bInterruptStarted S= bInterrupt AND astMotionStage[1].bBusy AND astMotionStage[2].bBusy AND astMotionStage[3].bBusy;
fbMove(
    astMotionStage:=astMotionStage,
    astPositionState:=astGoalPositions,
    nActiveMotorCount:=3,
    bExecute:=NOT bInterruptStarted,
);
IF fbMove.bDone OR tonTimer.Q OR (bInterruptStarted AND NOT fbMove.bBusy) THEN
    IF bInterrupt THEN
        AssertFalse(
            fbMove.bAtState,
            Message:='Should have been interrupted, but made it to the goal',
        );
    ELSE
        AssertTrue(
            fbMove.bAtState,
            Message:='Did not end at the state',
        );
        FOR nIter := 1 TO 3 DO
            AssertEquals_LREAL(
                Expected:=astGoalPositions[nIter].fPosition,
                Actual:=astMotionStage[nIter].stAxisStatus.fActPosition,
                Delta:=0.01,
                Message:='Did not reach the goal state',
            );
        END_FOR

    END_IF
    AssertFalse(
        fbMove.bBusy,
        Message:='Was busy while done',
    );
    AssertFalse(
        fbMove.bError,
        Message:='Should not end in error',
    );

    bOneTestDone := TRUE;
    TEST_FINISHED();
END_IF
END_METHOD

END_FUNCTION_BLOCK

// Tests/FB_PositionStateND_Test
FUNCTION_BLOCK FB_PositionStateND_Test EXTENDS FB_MotorTestSuite
(*
    Sanity checks for the following:
    - FB_PositionState1D
    - FB_PositionState2D
    - FB_PositionState3D
    The internals have already been tested, but we need to make sure that
    they've been put together at least somewhat sensibly.
    This FB will simply use each FB to move and check the results.

    Additional tests:
    - Regression test for issue #197 (input deadlock)
*)
VAR
    stMotionStage1: ST_MotionStage;
    stMotionStage2: ST_MotionStage;
    stMotionStage3: ST_MotionStage;
    astPositionState1: ARRAY[1..GeneralConstants.MAX_STATES] OF ST_PositionState;
    astPositionState2: ARRAY[1..GeneralConstants.MAX_STATES] OF ST_PositionState;
    astPositionState3: ARRAY[1..GeneralConstants.MAX_STATES] OF ST_PositionState;
    afbInternal: ARRAY[1..3] OF ARRAY[1..3] OF FB_PositionStateInternal;
    afbMotionStage: ARRAY[1..3] OF FB_MotionStage;

    fb_Move1D: FB_PositionState1D;
    fb_Move2D: FB_PositionState2D;
    fb_Move3D: FB_PositionState3D;

    nTestCounter: UINT;
    bOneTestDone: BOOL;
    fTestStartPos: LREAL;
    tonTimer: TON;
    nIter: DINT;
    bStatesReady: BOOL;

    eSetPos: E_TestStates;
    eGetPos: E_TestStates;
END_VAR


bStatesReady := TRUE;
FOR nIter := 1 TO 3 DO;
    astPositionState1[nIter].fPosition := nIter;
    astPositionState1[nIter].fDelta := 1;
    astPositionState1[nIter].fVelocity := 100;
    astPositionState2[nIter].fPosition := 10 + nIter;
    astPositionState2[nIter].fDelta := 1;
    astPositionState2[nIter].fVelocity := 100;
    astPositionState3[nIter].fPosition := 20 + nIter;
    astPositionState3[nIter].fDelta := 1;
    astPositionState3[nIter].fVelocity := 100;
    afbInternal[nIter][1](
        stMotionStage:=stMotionStage1,
        stPositionState:=astPositionState1[nIter],
    );
    afbInternal[nIter][2](
        stMotionStage:=stMotionStage2,
        stPositionState:=astPositionState2[nIter],
    );
    afbInternal[nIter][3](
        stMotionStage:=stMotionStage3,
        stPositionState:=astPositionState3[nIter],
    );
    SetGoodState(astPositionState1[nIter]);
    SetGoodState(astPositionState2[nIter]);
    SetGoodState(astPositionState3[nIter]);
    bStatesReady := bStatesReady AND astPositionState1[nIter].bUpdated;
    bStatesReady := bStatesReady AND astPositionState2[nIter].bUpdated;
    bStatesReady := bStatesReady AND astPositionState3[nIter].bUpdated;
END_FOR
SetEnables(stMotionStage1);
SetEnables(stMotionStage2);
SetEnables(stMotionStage3);
afbMotionStage[1](stMotionStage:=stMotionStage1);
afbMotionStage[2](stMotionStage:=stMotionStage2);
afbMotionStage[3](stMotionStage:=stMotionStage3);

IF bStatesReady AND nTestCounter = 0 THEN
    // Don't run any tests until the states are ready
    nTestCounter := 1;
    // Run all the motion FBs for one cycle to warm them up
    fb_Move1D(
        stMotionStage:=stMotionStage1,
        astPositionState:=astPositionState1,
        eEnumSet:=eSetPos,
        eEnumGet:=eGetPos,
        bEnable:=TRUE,
    );
    fb_Move2D(
        stMotionStage1:=stMotionStage1,
        stMotionStage2:=stMotionStage2,
        astPositionState1:=astPositionState1,
        astPositionState2:=astPositionState2,
        eEnumSet:=eSetPos,
        eEnumGet:=eGetPos,
        bEnable:=TRUE,
    );
    fb_Move3D(
        stMotionStage1:=stMotionStage1,
        stMotionStage2:=stMotionStage2,
        stMotionStage3:=stMotionStage3,
        astPositionState1:=astPositionState1,
        astPositionState2:=astPositionState2,
        astPositionState3:=astPositionState3,
        eEnumSet:=eSetPos,
        eEnumGet:=eGetPos,
        bEnable:=TRUE,
    );
END_IF

Test1D(1, E_TestStates.OUT);
Test1D(2, E_TestStates.TARGET1);
Test1D(3, E_TestStates.TARGET2);
Test2D(4, E_TestStates.OUT);
Test2D(5, E_TestStates.TARGET1);
Test2D(6, E_TestStates.TARGET2);
Test3D(7, E_TestStates.OUT);
Test3D(8, E_TestStates.TARGET1);
Test3D(9, E_TestStates.TARGET2);
TestInputDeadlock(10);

IF bOneTestDone THEN
    bOneTestDone := FALSE;
    nTestCounter := nTestCounter + 1;
    tonTimer(IN:=FALSE);
END_IF
// Use this timer to time out any tests that stall
tonTimer(
    IN:=bStatesReady,
    PT:=T#5s,
);

METHOD Test1D
VAR_INPUT
    nTestID: UINT;
    nState: E_TestStates;
END_VAR
VAR_INST
    nLocalInit: BOOL;
END_VAR

TEST(CONCAT('Test1D_state', DINT_TO_STRING(nState)));
IF nTestCounter <> nTestID THEN
    RETURN;
END_IF

IF NOT nLocalInit THEN
    eSetPos := nState;
    nLocalInit := TRUE;
END_IF

fb_Move1D(
    stMotionStage:=stMotionStage1,
    astPositionState:=astPositionState1,
    eEnumSet:=eSetPos,
    eEnumGet:=eGetPos,
    bEnable:=TRUE,
);
IF tonTimer.Q OR fb_Move1D.stPlcToEpics.bDone THEN
    AssertTrue(
        Condition:=fb_Move1D.stPlcToEpics.bDone,
        Message:='Done should be True after move',
    );
    AssertFalse(
        Condition:=fb_Move1D.stPlcToEpics.bBusy,
        Message:='Busy should be False after move',
    );
    AssertFalse(
        Condition:=fb_Move1D.stPlcToEpics.bError,
        Message:='Error should be False after move',
    );
    AssertEquals_DINT(
        Expected:=nState,
        Actual:=eGetPos,
        Message:='Did not get to the input state',
    );
    AssertEquals_LREAL(
        Expected:=astPositionState1[nState].fPosition,
        Actual:=stMotionStage1.stAxisStatus.fActPosition,
        Delta:=0.1,
        Message:='Did not get to the input state position',
    );
    fb_Move1D.stEpicsToPlc.bReset := TRUE;
    fb_Move1D(
        stMotionStage:=stMotionStage1,
        astPositionState:=astPositionState1,
        eEnumSet:=eSetPos,
        eEnumGet:=eGetPos,
        bEnable:=TRUE,
    );
    bOneTestDone := TRUE;
    nLocalInit := FALSE;
    TEST_FINISHED();
END_IF
END_METHOD

METHOD Test2D
VAR_INPUT
    nTestID: UINT;
    nState: E_TestStates;
END_VAR
VAR_INST
    nLocalInit: BOOL;
END_VAR

TEST(CONCAT('Test2D_state', DINT_TO_STRING(nState)));
IF nTestCounter <> nTestID THEN
    RETURN;
END_IF

IF NOT nLocalInit THEN
    eSetPos := nState;
    nLocalInit := TRUE;
END_IF

fb_Move2D(
    stMotionStage1:=stMotionStage1,
    stMotionStage2:=stMotionStage2,
    astPositionState1:=astPositionState1,
    astPositionState2:=astPositionState2,
    eEnumSet:=eSetPos,
    eEnumGet:=eGetPos,
    bEnable:=TRUE,
);
IF tonTimer.Q OR fb_Move2D.stPlcToEpics.bDone THEN
    AssertTrue(
        Condition:=fb_Move2D.stPlcToEpics.bDone,
        Message:='Done should be True after move',
    );
    AssertFalse(
        Condition:=fb_Move2D.stPlcToEpics.bBusy,
        Message:='Busy should be False after move',
    );
    AssertFalse(
        Condition:=fb_Move2D.stPlcToEpics.bError,
        Message:='Error should be False after move',
    );
    AssertEquals_DINT(
        Expected:=nState,
        Actual:=eGetPos,
        Message:='Did not get to the input state',
    );
    AssertEquals_LREAL(
        Expected:=astPositionState1[nState].fPosition,
        Actual:=stMotionStage1.stAxisStatus.fActPosition,
        Delta:=0.1,
        Message:='Did not get to the input state position for stage 1',
    );
    AssertEquals_LREAL(
        Expected:=astPositionState2[nState].fPosition,
        Actual:=stMotionStage2.stAxisStatus.fActPosition,
        Delta:=0.1,
        Message:='Did not get to the input state position for stage 2',
    );
    fb_Move2D.stEpicsToPlc.bReset := TRUE;
    fb_Move2D(
        stMotionStage1:=stMotionStage1,
        stMotionStage2:=stMotionStage2,
        astPositionState1:=astPositionState1,
        astPositionState2:=astPositionState2,
        eEnumSet:=eSetPos,
        eEnumGet:=eGetPos,
        bEnable:=TRUE,
    );
    bOneTestDone := TRUE;
    nLocalInit := FALSE;
    TEST_FINISHED();
END_IF
END_METHOD

METHOD Test3D
VAR_INPUT
    nTestID: UINT;
    nState: E_TestStates;
END_VAR
VAR_INST
    nLocalInit: BOOL;
END_VAR

TEST(CONCAT('Test3D_state', DINT_TO_STRING(nState)));
IF nTestCounter <> nTestID THEN
    RETURN;
END_IF

IF NOT nLocalInit THEN
    eSetPos := nState;
    nLocalInit := TRUE;
END_IF

fb_Move3D(
    stMotionStage1:=stMotionStage1,
    stMotionStage2:=stMotionStage2,
    stMotionStage3:=stMotionStage3,
    astPositionState1:=astPositionState1,
    astPositionState2:=astPositionState2,
    astPositionState3:=astPositionState3,
    eEnumSet:=eSetPos,
    eEnumGet:=eGetPos,
    bEnable:=TRUE,
);
IF tonTimer.Q OR fb_Move3D.stPlcToEpics.bDone THEN
    AssertTrue(
        Condition:=fb_Move3D.stPlcToEpics.bDone,
        Message:='Done should be True after move',
    );
    AssertFalse(
        Condition:=fb_Move3D.stPlcToEpics.bBusy,
        Message:='Busy should be False after move',
    );
    AssertFalse(
        Condition:=fb_Move3D.stPlcToEpics.bError,
        Message:='Error should be False after move',
    );
    AssertEquals_DINT(
        Expected:=nState,
        Actual:=eGetPos,
        Message:='Did not get to the input state',
    );
    AssertEquals_LREAL(
        Expected:=astPositionState1[nState].fPosition,
        Actual:=stMotionStage1.stAxisStatus.fActPosition,
        Delta:=0.1,
        Message:='Did not get to the input state position for stage 1',
    );
    AssertEquals_LREAL(
        Expected:=astPositionState2[nState].fPosition,
        Actual:=stMotionStage2.stAxisStatus.fActPosition,
        Delta:=0.1,
        Message:='Did not get to the input state position for stage 2',
    );
    AssertEquals_LREAL(
        Expected:=astPositionState3[nState].fPosition,
        Actual:=stMotionStage3.stAxisStatus.fActPosition,
        Delta:=0.1,
        Message:='Did not get to the input state position for stage 3',
    );
    fb_Move3D.stEpicsToPlc.bReset := TRUE;
    fb_Move3D(
        stMotionStage1:=stMotionStage1,
        stMotionStage2:=stMotionStage2,
        stMotionStage3:=stMotionStage3,
        astPositionState1:=astPositionState1,
        astPositionState2:=astPositionState2,
        astPositionState3:=astPositionState3,
        eEnumSet:=eSetPos,
        eEnumGet:=eGetPos,
        bEnable:=TRUE,
    );
    bOneTestDone := TRUE;
    nLocalInit := FALSE;
    TEST_FINISHED();
END_IF
END_METHOD

METHOD TestInputDeadlock
(*
    Regression test for issue #197

    How to reproduce the issue:
    1. Get the function block into any motion error
    2. Ask for a move while in the error state

    Then, the state mover never moves again.

    To test we will follow steps 1 and 2, then reset the error, then move.

    With our fix, our second attempt at the move (after an error reset) will succeed.
    Our first attempt will fail regardless, since you cannot move a motor that is in an error state.

    Without our fix, the motor could never be moved ever again and this move will time out.
*)
VAR_INPUT
    nTestID: UINT;
END_VAR
VAR_INST
    nTestStep: UINT := 1;
    eNewGoal: E_TestStates;
END_VAR

TEST('TestInputDeadlock');
IF nTestCounter <> nTestID THEN
    RETURN;
END_IF

CASE nTestStep OF
    // Step 1: Normal move
    1:
        // Normal move: pick any other state
        IF eGetPos = E_TestStates.OUT THEN
            eNewGoal := E_TestStates.TARGET1;
        ELSE
            eNewGoal := E_TestStates.OUT;
        END_IF
        eSetPos := eNewGoal;
        nTestStep := 2;
    // Step 2: Cause a motion error. Easiest is to just set bError to TRUE during a move.
    2:
        // Cause the error if it's time
        IF stMotionStage1.bBusy THEN
            stMotionStage1.bError := TRUE;
            stMotionStage1.nErrorId := 16#4FFF;
        ELSIF stMotionStage1.bError THEN
            nTestStep := 3;
        END_IF
     // Step 3: another normal move. This should get us into the potential bugged state.
     3:
        eSetPos := eNewGoal;
        nTestStep := 4;
    // Step 4: reset the error, which will allow fixed versions of the code to resume normal operations.
    4:
        fb_Move1D.stEpicsToPlc.bReset := TRUE;
        IF NOT stMotionStage1.bError THEN
            nTestStep := 5;
        END_IF
    // Step 5: last normal move, which will succeed if we fixed the bug.
    5:
        eSetPos := eNewGoal;
        IF eGetPos = E_TestStates.Unknown THEN
            nTestStep := 6;
        END_IF
    // Step 6: wait for the move to finish
    6:
        IF eGetPos = eNewGoal THEN
            nTestStep := 7;
        END_IF
END_CASE

fb_Move1D(
    stMotionStage:=stMotionStage1,
    astPositionState:=astPositionState1,
    eEnumSet:=eSetPos,
    eEnumGet:=eGetPos,
    bEnable:=TRUE,
);

// Timeout and checks
IF tonTimer.Q OR nTestStep = 7 THEN
    AssertFalse(
        tonTimer.Q,
        'Timeout in deadlock test',
    );
    AssertEquals_UINT(
        Expected:=eNewGoal,
        Actual:=eGetPos,
        'Did not reach a goal state in deadlock test',
    );
    fb_Move1D.stEpicsToPlc.bReset := TRUE;
    fb_Move1D(
        stMotionStage:=stMotionStage1,
        astPositionState:=astPositionState1,
        eEnumSet:=eSetPos,
        eEnumGet:=eGetPos,
        bEnable:=TRUE,
    );
    bOneTestDone := TRUE;
    TEST_FINISHED();
END_IF
END_METHOD

END_FUNCTION_BLOCK

// Tests/FB_PositionStatePMPSND_Test
FUNCTION_BLOCK FB_PositionStatePMPSND_Test EXTENDS FB_MotorTestSuite
(*
    Sanity checks for the following:
    - FB_PositionStatePMPS1D
    - FB_PositionStatePMPS2D
    - FB_PositionStatePMPS3D
    The internals have already been tested, but we need to make sure that
    they've been put together at least somewhat sensibly.
    This FB will simply use each FB to move and check the results.
    In addition to reaching the goals, we need to check the beam assertions
    and the pmps limit enables.
*)
VAR
    stMotionStage1: ST_MotionStage;
    stMotionStage2: ST_MotionStage;
    stMotionStage3: ST_MotionStage;
    astPositionState1: ARRAY[1..GeneralConstants.MAX_STATES] OF ST_PositionState;
    astPositionState2: ARRAY[1..GeneralConstants.MAX_STATES] OF ST_PositionState;
    astPositionState3: ARRAY[1..GeneralConstants.MAX_STATES] OF ST_PositionState;
    afbInternal: ARRAY[1..3] OF ARRAY[1..3] OF FB_PositionStateInternal;
    afbMotionStage: ARRAY[1..3] OF FB_MotionStage;

    astBeam: ARRAY[0..3] OF ST_DbStateParams;

    fb_Move1D: FB_PositionStatePMPS1D;
    fb_Move2D: FB_PositionStatePMPS2D;
    fb_Move3D: FB_PositionStatePMPS3D;

    nTestCounter: UINT;
    bOneTestDone: BOOL;
    fTestStartPos: LREAL;
    tonTimer: TON;
    nIter: DINT;
    bStatesReady: BOOL;

    eSetPos: E_TestStates;
    eGetPos: E_TestStates;

    fbArbiter1D: FB_Arbiter(1);
    fbArbiter2D: FB_Arbiter(2);
    fbArbiter3D: FB_Arbiter(3);

    fbSubSysIO1D: FB_DummyArbIO;
    fbSubSysIO2D: FB_DummyArbIO;
    fbSubSysIO3D: FB_DummyArbIO;

    jsonHelper: FB_PMPSJsonTestHelper;
END_VAR


bStatesReady := TRUE;
FOR nIter := 1 TO 3 DO;
    astPositionState1[nIter].fPosition := nIter;
    astPositionState1[nIter].fDelta := 0.5;
    astPositionState1[nIter].fVelocity := 100;
    SetGoodState(astPositionState1[nIter]);
    astPositionState2[nIter].fPosition := 10 + nIter;
    astPositionState2[nIter].fDelta := 0.5;
    astPositionState2[nIter].fVelocity := 100;
    SetGoodState(astPositionState2[nIter]);
    astPositionState3[nIter].fPosition := 20 + nIter;
    astPositionState3[nIter].fDelta := 0.5;
    astPositionState3[nIter].fVelocity := 100;
    SetGoodState(astPositionState3[nIter]);
    afbInternal[nIter][1](
        stMotionStage:=stMotionStage1,
        stPositionState:=astPositionState1[nIter],
    );
    afbInternal[nIter][2](
        stMotionStage:=stMotionStage2,
        stPositionState:=astPositionState2[nIter],
    );
    afbInternal[nIter][3](
        stMotionStage:=stMotionStage3,
        stPositionState:=astPositionState3[nIter],
    );
    bStatesReady := bStatesReady AND astPositionState1[nIter].bUpdated;
    bStatesReady := bStatesReady AND astPositionState2[nIter].bUpdated;
    bStatesReady := bStatesReady AND astPositionState3[nIter].bUpdated;
END_FOR
SetEnablesPMPS(stMotionStage1);
SetEnablesPMPS(stMotionStage2);
SetEnablesPMPS(stMotionStage3);
IF nTestCounter <= 3 THEN
    // Startup tests, make sure the motor is enabled so we can inspect MC_Power's output
    // Otherwise we can't snoop on the PlcToNc control DWORD since this is all 0's if disabled
    // When enabled, some of the other bits go to 1 to represent directional enables
    stMotionStage1.nEnableMode := E_StageEnableMode.ALWAYS;
    stMotionStage2.nEnableMode := E_StageEnableMode.ALWAYS;
    stMotionStage3.nEnableMode := E_StageEnableMode.ALWAYS;
ELSE
    // Otherwise, make sure the most complicated mode (and the default) works
    stMotionStage1.nEnableMode := E_StageEnableMode.DURING_MOTION;
    stMotionStage2.nEnableMode := E_StageEnableMode.DURING_MOTION;
    stMotionStage3.nEnableMode := E_StageEnableMode.DURING_MOTION;
END_IF
afbMotionStage[1](stMotionStage:=stMotionStage1);
afbMotionStage[2](stMotionStage:=stMotionStage2);
afbMotionStage[3](stMotionStage:=stMotionStage3);

astBeam[E_TestStates.Unknown].stBeamParams := PMPS_GVL.cst0RateBeam;
astBeam[E_TestStates.Unknown].nRequestAssertionID := 1;
astBeam[E_TestStates.Unknown].sPmpsState := 'trans';
astBeam[E_TestStates.OUT].stBeamParams := PMPS_GVL.cstFullBeam;
astBeam[E_TestStates.OUT].nRequestAssertionID := 2;
astBeam[E_TestStates.OUT].sPmpsState := 'out';
astBeam[E_TestStates.TARGET1].stBeamParams := PMPS_GVL.cstFullBeam;
astBeam[E_TestStates.TARGET1].stBeamParams.nTran := 0.1;
astBeam[E_TestStates.TARGET1].nRequestAssertionID := 3;
astBeam[E_TestStates.TARGET1].sPmpsState := 'target1';
astBeam[E_TestStates.TARGET2].stBeamParams := PMPS_GVL.cstFullBeam;
astBeam[E_TestStates.TARGET2].stBeamParams.nTran := 0.01;
astBeam[E_TestStates.TARGET2].nRequestAssertionID := 4;
astBeam[E_TestStates.TARGET2].sPmpsState := 'target2';

// Assign beam params to states 1
astPositionState1[E_TestStates.OUT].stPMPS := astBeam[E_TestStates.OUT];
astPositionState1[E_TestStates.TARGET1].stPMPS := astBeam[E_TestStates.TARGET1];
astPositionState1[E_TestStates.TARGET2].stPMPS := astBeam[E_TestStates.TARGET2];

// Set some names for maybe help in debug
astPositionState1[E_TestStates.OUT].sName := 'OUT';
astPositionState1[E_TestStates.TARGET1].sName := 'TARGET1';
astPositionState1[E_TestStates.TARGET2].sName := 'TARGET2';
astPositionState2[E_TestStates.OUT].sName := 'OUT';
astPositionState2[E_TestStates.TARGET1].sName := 'TARGET1';
astPositionState2[E_TestStates.TARGET2].sName := 'TARGET2';
astPositionState3[E_TestStates.OUT].sName := 'OUT';
astPositionState3[E_TestStates.TARGET1].sName := 'TARGET1';
astPositionState3[E_TestStates.TARGET2].sName := 'TARGET2';

// Load a fake json doc to be consumed by our FB
jsonHelper(
    astBeamParams:=astBeam,
    bExecute:=TRUE,
    sDevName:='test',
);

IF bStatesReady AND nTestCounter = 0 THEN
    // Don't run any tests until the states are ready
    nTestCounter := 1;
END_IF

TestStartup1D(1);
TestStartup2D(2);
TestStartup3D(3);
Test1D(4, E_TestStates.OUT);
Test1D(5, E_TestStates.TARGET1);
Test1D(6, E_TestStates.TARGET2);
Test2D(7, E_TestStates.OUT);
Test2D(8, E_TestStates.TARGET1);
Test2D(9, E_TestStates.TARGET2);
Test3D(10, E_TestStates.OUT);
Test3D(11, E_TestStates.TARGET1);
Test3D(12, E_TestStates.TARGET2);

IF bOneTestDone THEN
    bOneTestDone := FALSE;
    nTestCounter := nTestCounter + 1;
    tonTimer(IN:=FALSE);
END_IF
// Use this timer to time out any tests that stall
tonTimer(
    IN:=bStatesReady,
    PT:=T#5s,
);

METHOD AssertMotionLims: BOOL
VAR_IN_OUT
    stMotionStage: ST_MotionStage;
    astPositionState: ARRAY[1..GeneralConstants.MAX_STATES] OF ST_PositionState;
END_VAR
VAR_INPUT
    eState: E_TestStates;
    sID: STRING;
END_VAR
VAR
    nExpected: DWORD;
END_VAR

IF F_AtPositionState(stMotionStage, astPositionState[eState]) THEN
    // Both allowed
    nExpected := 2#111;
ELSIF stMotionStage.stAxisStatus.fActPosition < astPositionState[eState].fPosition THEN
    // Only + allowed
    nExpected := 2#011;
ELSE
    // Only - allowed
    nExpected := 2#101;
END_IF

IF stMotionStage.Axis.PlcToNc.ControlDWord > 0 THEN
    AssertEquals_DWORD(
        Expected:=nExpected,
        Actual:=stMotionStage.Axis.PlcToNc.ControlDWord,
        Message:=CONCAT('Wrong control dword in test ', sID),
    );
    AssertMotionLims := TRUE;
END_IF
END_METHOD

METHOD Test1D
VAR_INPUT
    nTestID: UINT;
    eState: E_TestStates;
END_VAR
VAR_INST
    fbFFHWO: FB_HardwareFFOutput;
    bInit: BOOL;
    bLimAsserted: BOOL;
END_VAR

TEST(CONCAT('Test1D_state', UINT_TO_STRING(eState)));
IF nTestCounter <> nTestID THEN
    RETURN;
END_IF

IF NOT bInit THEN
    eSetPos := eState;
END_IF

fbSubSysIO1D(
    LA:=fbArbiter1D,
    FFO:=fbFFHWO,
);

fb_Move1D(
    stMotionStage:=stMotionStage1,
    astPositionState:=astPositionState1,
    eEnumSet:=eSetPos,
    eEnumGet:=eGetPos,
    fbFFHWO:=fbFFHWO,
    fbArbiter:=fbArbiter1D,
    bEnableMotion:=TRUE,
    bEnableBeamParams:=TRUE,
    bEnablePositionLimits:=TRUE,
    bReadDBNow:=NOT bInit,
    sDeviceName:='test',
    sTransitionKey:='trans',
);

// When ready: check that directonal enables are correct
bLimAsserted S= AssertMotionLims(stMotionStage1, astPositionState1, eState, CONCAT('1D mot 1 state ', UINT_TO_STRING(eState)));


IF NOT bInit THEN
    bInit := TRUE;
END_IF

IF tonTimer.Q OR fb_Move1D.stPlcToEpics.bDone THEN
    AssertTrue(
        bLimAsserted,
        'Skipped limit assert test',
    );
    AssertTrue(
        Condition:=fb_Move1D.stPlcToEpics.bDone,
        Message:='Done should be True after move',
    );
    AssertFalse(
        Condition:=fb_Move1D.stPlcToEpics.bBusy,
        Message:='Busy should be False after move',
    );
    AssertFalse(
        Condition:=fb_Move1D.stPlcToEpics.bError,
        Message:='Error should be False after move',
    );
    AssertEquals_UINT(
        Expected:=eState,
        Actual:=eGetPos,
        Message:='Did not get to the input state',
    );
    AssertEquals_LREAL(
        Expected:=astPositionState1[eState].fPosition,
        Actual:=stMotionStage1.stAxisStatus.fActPosition,
        Delta:=0.1,
        Message:='Did not get to the input state position',
    );
    AssertTrue(
        fbArbiter1D.CheckRequestInPool(astBeam[eState].nRequestAssertionID),
        'Destination bp should have been in the arbiter',
    );
    fb_Move1D.stEpicsToPlc.bReset := TRUE;
    fb_Move1D(
        stMotionStage:=stMotionStage1,
        astPositionState:=astPositionState1,
        eEnumSet:=eSetPos,
        eEnumGet:=eGetPos,
        fbFFHWO:=fbFFHWO,
        fbArbiter:=fbArbiter1D,
        bEnableMotion:=TRUE,
        bEnableBeamParams:=TRUE,
        bEnablePositionLimits:=TRUE,
    );
    bInit := FALSE;
    bLimAsserted := FALSE;
    bOneTestDone := TRUE;
    TEST_FINISHED();
END_IF
END_METHOD

METHOD Test2D
VAR_INPUT
    nTestID: UINT;
    eState: E_TestStates;
END_VAR
VAR_INST
    fbFFHWO: FB_HardwareFFOutput;
    bInit: BOOL;
    bLimAsserted1: BOOL;
    bLimAsserted2: BOOL;
END_VAR

TEST(CONCAT('Test2D_state', UINT_TO_STRING(eState)));
IF nTestCounter <> nTestID THEN
    RETURN;
END_IF

IF NOT bInit THEN
    eSetPos := eState;
END_IF

fbSubSysIO2D(
    LA:=fbArbiter2D,
    FFO:=fbFFHWO,
);

fb_Move2D(
    stMotionStage1:=stMotionStage1,
    stMotionStage2:=stMotionStage2,
    astPositionState1:=astPositionState1,
    astPositionState2:=astPositionState2,
    eEnumSet:=eSetPos,
    eEnumGet:=eGetPos,
    fbFFHWO:=fbFFHWO,
    fbArbiter:=fbArbiter2D,
    bEnableMotion:=TRUE,
    bEnableBeamParams:=TRUE,
    bEnablePositionLimits:=TRUE,
    bReadDBNow:=NOT bInit,
    sDeviceName:='test',
    sTransitionKey:='trans',
);

// When ready: check that directonal enables are correct
bLimAsserted1 S= AssertMotionLims(stMotionStage1, astPositionState1, eState, CONCAT('2D mot 1 state ', UINT_TO_STRING(eState)));
bLimAsserted2 S= AssertMotionLims(stMotionStage2, astPositionState2, eState, CONCAT('2D mot 2 state ', UINT_TO_STRING(eState)));

IF NOT bInit THEN
    bInit := TRUE;
END_IF

IF tonTimer.Q OR fb_Move2D.stPlcToEpics.bDone THEN
    AssertTrue(
        bLimAsserted1 AND bLimAsserted2,
        'Skipped limit assert test',
    );
    AssertTrue(
        Condition:=fb_Move2D.stPlcToEpics.bDone,
        Message:='Done should be True after move',
    );
    AssertFalse(
        Condition:=fb_Move2D.stPlcToEpics.bBusy,
        Message:='Busy should be False after move',
    );
    AssertFalse(
        Condition:=fb_Move2D.stPlcToEpics.bError,
        Message:='Error should be False after move',
    );
    AssertEquals_UINT(
        Expected:=eState,
        Actual:=eGetPos,
        Message:='Did not get to the input state',
    );
    AssertEquals_LREAL(
        Expected:=astPositionState1[eState].fPosition,
        Actual:=stMotionStage1.stAxisStatus.fActPosition,
        Delta:=0.1,
        Message:='Did not get to the input state position',
    );
    AssertEquals_LREAL(
        Expected:=astPositionState2[eState].fPosition,
        Actual:=stMotionStage2.stAxisStatus.fActPosition,
        Delta:=0.1,
        Message:='Did not get to the input state position',
    );
    AssertTrue(
        fbArbiter2D.CheckRequestInPool(astBeam[eState].nRequestAssertionID),
        'Destination bp should have been in the arbiter',
    );
    fb_Move2D.stEpicsToPlc.bReset := TRUE;
    fb_Move2D(
        stMotionStage1:=stMotionStage1,
        stMotionStage2:=stMotionStage2,
        astPositionState1:=astPositionState1,
        astPositionState2:=astPositionState2,
        eEnumSet:=eSetPos,
        eEnumGet:=eGetPos,
        fbFFHWO:=fbFFHWO,
        fbArbiter:=fbArbiter2D,
        bEnableMotion:=TRUE,
        bEnableBeamParams:=TRUE,
        bEnablePositionLimits:=TRUE,
    );
    bInit := FALSE;
    bLimAsserted1 := FALSE;
    bLimAsserted2 := FALSE;
    bOneTestDone := TRUE;
    TEST_FINISHED();
END_IF
END_METHOD

METHOD Test3D
VAR_INPUT
    nTestID: UINT;
    eState: E_TestStates;
END_VAR
VAR_INST
    fbFFHWO: FB_HardwareFFOutput;
    bInit: BOOL;
    bLimAsserted1: BOOL;
    bLimAsserted2: BOOL;
    bLimAsserted3: BOOL;
END_VAR

TEST(CONCAT('Test3D_state', UINT_TO_STRING(eState)));
IF nTestCounter <> nTestID THEN
    RETURN;
END_IF

IF NOT bInit THEN
    eSetPos := eState;
END_IF

fbSubSysIO3D(
    LA:=fbArbiter3D,
    FFO:=fbFFHWO,
);

fb_Move3D(
    stMotionStage1:=stMotionStage1,
    stMotionStage2:=stMotionStage2,
    stMotionStage3:=stMotionStage3,
    eEnumSet:=eSetPos,
    eEnumGet:=eGetPos,
    astPositionState1:=astPositionState1,
    astPositionState2:=astPositionState2,
    astPositionState3:=astPositionState3,
    fbFFHWO:=fbFFHWO,
    fbArbiter:=fbArbiter3D,
    bEnableMotion:=TRUE,
    bEnableBeamParams:=TRUE,
    bEnablePositionLimits:=TRUE,
    bReadDBNow:=NOT bInit,
    sDeviceName:='test',
    sTransitionKey:='trans',
);

// When ready: check that directonal enables are correct
bLimAsserted1 S= AssertMotionLims(stMotionStage1, astPositionState1, eState, CONCAT('3D mot 1 state ', UINT_TO_STRING(eState)));
bLimAsserted2 S= AssertMotionLims(stMotionStage2, astPositionState2, eState, CONCAT('3D mot 2 state ', UINT_TO_STRING(eState)));
bLimAsserted3 S= AssertMotionLims(stMotionStage3, astPositionState3, eState, CONCAT('3D mot 3 state ', UINT_TO_STRING(eState)));

IF NOT bInit THEN
    bInit := TRUE;
END_IF

IF tonTimer.Q OR fb_Move3D.stPlcToEpics.bDone THEN
    AssertTrue(
        bLimAsserted1 AND bLimAsserted2 AND bLimAsserted3,
        'Skipped limit assert test',
    );
    AssertTrue(
        Condition:=fb_Move3D.stPlcToEpics.bDone,
        Message:='Done should be True after move',
    );
    AssertFalse(
        Condition:=fb_Move3D.stPlcToEpics.bBusy,
        Message:='Busy should be False after move',
    );
    AssertFalse(
        Condition:=fb_Move3D.stPlcToEpics.bError,
        Message:='Error should be False after move',
    );
    AssertEquals_UINT(
        Expected:=eState,
        Actual:=eGetPos,
        Message:='Did not get to the input state',
    );
    AssertEquals_LREAL(
        Expected:=astPositionState1[eState].fPosition,
        Actual:=stMotionStage1.stAxisStatus.fActPosition,
        Delta:=0.1,
        Message:='Did not get to the input state position',
    );
    AssertEquals_LREAL(
        Expected:=astPositionState2[eState].fPosition,
        Actual:=stMotionStage2.stAxisStatus.fActPosition,
        Delta:=0.1,
        Message:='Did not get to the input state position',
    );
    AssertEquals_LREAL(
        Expected:=astPositionState3[eState].fPosition,
        Actual:=stMotionStage3.stAxisStatus.fActPosition,
        Delta:=0.1,
        Message:='Did not get to the input state position',
    );
    AssertTrue(
        fbArbiter3D.CheckRequestInPool(astBeam[eState].nRequestAssertionID),
        'Destination bp should have been in the arbiter',
    );
    fb_Move3D.stEpicsToPlc.bReset := TRUE;
    fb_Move3D(
        stMotionStage1:=stMotionStage1,
        stMotionStage2:=stMotionStage2,
        stMotionStage3:=stMotionStage3,
        astPositionState1:=astPositionState1,
        astPositionState2:=astPositionState2,
        astPositionState3:=astPositionState3,
        eEnumSet:=eSetPos,
        eEnumGet:=eGetPos,
        fbFFHWO:=fbFFHWO,
        fbArbiter:=fbArbiter3D,
        bEnableMotion:=TRUE,
        bEnableBeamParams:=TRUE,
        bEnablePositionLimits:=TRUE,
    );
    bInit := FALSE;
    bLimAsserted1 := FALSE;
    bLimAsserted2 := FALSE;
    bLimAsserted3 := FALSE;
    bOneTestDone := TRUE;
    TEST_FINISHED();
END_IF
END_METHOD

METHOD TestStartup1D
(*
    - On startup, there should be no move request
    - In this case, we start in an unknown state since (0, 0, 0) is not matching any state for any motor
    - Movement should be free but the transition assertion must be active
*)
VAR_INPUT
    nTestID: UINT;
END_VAR
VAR_INST
    fbFFHWO: FB_HardwareFFOutput;
    bInit: BOOL;
END_VAR

TEST('TestStartup1D');
IF nTestCounter <> nTestID THEN
    RETURN;
END_IF

fb_Move1D(
    stMotionStage:=stMotionStage1,
    astPositionState:=astPositionState1,
    eEnumSet:=eSetPos,
    eEnumGet:=eGetPos,
    fbFFHWO:=fbFFHWO,
    fbArbiter:=fbArbiter1D,
    bEnableMotion:=TRUE,
    bEnableBeamParams:=TRUE,
    bEnablePositionLimits:=TRUE,
    bReadDBNow:=NOT bInit,
    sDeviceName:='test',
    sTransitionKey:='trans',
);

bInit := TRUE;

// We sit in this fb for some timeout number of seconds on purpose, not an error
IF tonTimer.Q THEN
    // We should neither be busy nor done (we didn't do anything)
    AssertFalse(
        Condition:=fb_Move1D.stPlcToEpics.bDone,
        Message:='Done should be False with no move',
    );
    AssertFalse(
        Condition:=fb_Move1D.stPlcToEpics.bBusy,
        Message:='Busy should be False with no move',
    );
    // We should still be at 0,0,0
    AssertEquals_LREAL(
        Expected:=0,
        Actual:=stMotionStage1.stAxisStatus.fActPosition,
        Delta:=0.0001,
        Message:='Why did we move? motor1 should have default position',
    );
    // We should be able to move both directions, which is control word 7 (2#111)
    AssertEquals_DWORD(
        Expected:=2#111,
        Actual:=stMotionStage1.Axis.PlcToNc.ControlDWord,
        Message:='Expected full +/- enables',
    );
    AssertTrue(
        fbArbiter1D.CheckRequestInPool(astBeam[E_TestStates.Unknown].nRequestAssertionID),
        'Transition assertion ID not in pool',
    );
    bOneTestDone := TRUE;
    TEST_FINISHED();
END_IF
END_METHOD

METHOD TestStartup2D
(*
    - On startup, there should be no move request
    - Starting from (0, 0, 0) all motors should only be allowed to move +
*)
VAR_INPUT
    nTestID: UINT;
END_VAR
VAR_INST
    fbFFHWO: FB_HardwareFFOutput;
    bInit: BOOL;
END_VAR

TEST('TestStartup2D');
IF nTestCounter <> nTestID THEN
    RETURN;
END_IF

fb_Move2D(
    stMotionStage1:=stMotionStage1,
    stMotionStage2:=stMotionStage2,
    astPositionState1:=astPositionState1,
    astPositionState2:=astPositionState2,
    eEnumSet:=eSetPos,
    eEnumGet:=eGetPos,
    fbFFHWO:=fbFFHWO,
    fbArbiter:=fbArbiter2D,
    bEnableMotion:=TRUE,
    bEnableBeamParams:=TRUE,
    bEnablePositionLimits:=TRUE,
    bReadDBNow:=NOT bInit,
    sDeviceName:='test',
    sTransitionKey:='trans',
);

bInit := TRUE;

// We sit in this fb for some timeout number of seconds on purpose, not an error
IF tonTimer.Q THEN
    // We should neither be busy nor done (we didn't do anything)
    AssertFalse(
        Condition:=fb_Move2D.stPlcToEpics.bDone,
        Message:='Done should be False with no move',
    );
    AssertFalse(
        Condition:=fb_Move2D.stPlcToEpics.bBusy,
        Message:='Busy should be False with no move',
    );
    // We should still be at 0,0,0
    AssertEquals_LREAL(
        Expected:=0,
        Actual:=stMotionStage1.stAxisStatus.fActPosition,
        Delta:=0.0001,
        Message:='Why did we move? motor1 should have default position',
    );
    AssertEquals_LREAL(
        Expected:=0,
        Actual:=stMotionStage2.stAxisStatus.fActPosition,
        Delta:=0.0001,
        Message:='Why did we move? motor2 should have default position',
    );
    // We should be able to move both directions, which is control word 7 (2#111)
    AssertEquals_DWORD(
        Expected:=2#111,
        Actual:=stMotionStage1.Axis.PlcToNc.ControlDWord,
        Message:='Expected full +/- enables',
    );
    AssertEquals_DWORD(
        Expected:=2#111,
        Actual:=stMotionStage2.Axis.PlcToNc.ControlDWord,
        Message:='Expected full +/- enables',
    );
    AssertTrue(
        fbArbiter2D.CheckRequestInPool(astBeam[E_TestStates.Unknown].nRequestAssertionID),
        'Transition assertion ID not in pool',
    );
    bOneTestDone := TRUE;
    TEST_FINISHED();
END_IF
END_METHOD

METHOD TestStartup3D
(*
    - On startup, there should be no move request
    - Starting from (0, 0, 0) all motors should only be allowed to move +
*)
VAR_INPUT
    nTestID: UINT;
END_VAR
VAR_INST
    fbFFHWO: FB_HardwareFFOutput;
    bInit: BOOL;
END_VAR

TEST('TestStartup3D');
IF nTestCounter <> nTestID THEN
    RETURN;
END_IF

fb_Move3D(
    stMotionStage1:=stMotionStage1,
    stMotionStage2:=stMotionStage2,
    stMotionStage3:=stMotionStage3,
    astPositionState1:=astPositionState1,
    astPositionState2:=astPositionState2,
    astPositionState3:=astPositionState3,
    eEnumSet:=eSetPos,
    eEnumGet:=eGetPos,
    fbFFHWO:=fbFFHWO,
    fbArbiter:=fbArbiter3D,
    bEnableMotion:=TRUE,
    bEnableBeamParams:=TRUE,
    bEnablePositionLimits:=TRUE,
    bReadDBNow:=NOT bInit,
    sDeviceName:='test',
    sTransitionKey:='trans',
);

bInit := TRUE;

// We sit in this fb for some timeout number of seconds on purpose, not an error
IF tonTimer.Q THEN
    // We should neither be busy nor done (we didn't do anything)
    AssertFalse(
        Condition:=fb_Move3D.stPlcToEpics.bDone,
        Message:='Done should be False with no move',
    );
    AssertFalse(
        Condition:=fb_Move3D.stPlcToEpics.bBusy,
        Message:='Busy should be False with no move',
    );
    // We should still be at 0,0,0
    AssertEquals_LREAL(
        Expected:=0,
        Actual:=stMotionStage1.stAxisStatus.fActPosition,
        Delta:=0.0001,
        Message:='Why did we move? motor1 should have default position',
    );
    AssertEquals_LREAL(
        Expected:=0,
        Actual:=stMotionStage2.stAxisStatus.fActPosition,
        Delta:=0.0001,
        Message:='Why did we move? motor2 should have default position',
    );
    AssertEquals_LREAL(
        Expected:=0,
        Actual:=stMotionStage3.stAxisStatus.fActPosition,
        Delta:=0.0001,
        Message:='Why did we move? motor3 should have default position',
    );
    // We should be able to move both directions, which is control word 7 (2#111)
    AssertEquals_DWORD(
        Expected:=2#111,
        Actual:=stMotionStage1.Axis.PlcToNc.ControlDWord,
        Message:='Expected full +/- enables',
    );
    AssertEquals_DWORD(
        Expected:=2#111,
        Actual:=stMotionStage2.Axis.PlcToNc.ControlDWord,
        Message:='Expected full +/- enables',
    );
    AssertEquals_DWORD(
        Expected:=2#111,
        Actual:=stMotionStage3.Axis.PlcToNc.ControlDWord,
        Message:='Expected full +/- enables',
    );
    AssertTrue(
        fbArbiter3D.CheckRequestInPool(astBeam[E_TestStates.Unknown].nRequestAssertionID),
        'Transition assertion ID not in pool',
    );
    bOneTestDone := TRUE;
    TEST_FINISHED();
END_IF
END_METHOD

END_FUNCTION_BLOCK

// Tests/FB_PositionStateRead_Test
FUNCTION_BLOCK FB_PositionStateRead_Test EXTENDS TcUnit.FB_TestSuite
(*
    Test that FB_PositionStateRead works exactly how it should
    according to its API during normal and failure states.
*)
VAR
    stMotionStage: ST_MotionStage;
    fbMotionStage: FB_MotionStage;
    astPositionState: ARRAY[1..GeneralConstants.MAX_STATES] OF ST_PositionState;
    afbInternal: ARRAY[1..3] OF FB_PositionStateInternal;
    stDummyPos: ST_PositionState;
    fbTestMove: FB_TestHelperSetAndMove;
    fbRead: FB_PositionStateRead;

    nTestCounter: UINT;
    bOneTestDone: BOOL;
    fTestStartPos: LREAL;
    tonTimer: TON;
    nIter: DINT;
    bStatesReady: BOOL;
END_VAR


astPositionState[1].sName := 'UNO';
astPositionState[1].fPosition := 10;
astPositionState[1].fDelta := 1;
astPositionState[1].bValid := TRUE;
astPositionState[1].bUseRawCounts := FALSE;

astPositionState[2].sName := 'DOS';
astPositionState[2].fPosition := 20;
astPositionState[2].fDelta := 1;
astPositionState[2].bValid := FALSE;
astPositionState[2].bUseRawCounts := FALSE;

astPositionState[3].sName := 'TRES';
astPositionState[3].fPosition := 30;
astPositionState[3].fDelta := 1;
astPositionState[3].bValid := TRUE;
astPositionState[3].bUseRawCounts := FALSE;

astPositionState[4].sName := 'QUATRO';
astPositionState[4].fPosition := 30;
astPositionState[4].fDelta := 1;
astPositionState[4].bValid := FALSE;
astPositionState[4].bUseRawCounts := FALSE;

bStatesReady := TRUE;
FOR nIter := 1 TO 4 DO
    afbInternal[nIter](
        stMotionStage:=stMotionStage,
        stPositionState:=astPositionState[nIter],
    );
    bStatesReady := bStatesReady AND astPositionState[nIter].bUpdated;
END_FOR
fbMotionStage(stMotionStage:=stMotionStage);

// At position 1 check
TestStaticPosition(
    nTestIndex:=0,
    sTestName:='AtPos1',
    fPosition:=astPositionState[1].fPosition + 0.2 * astPositionState[1].fDelta,
    bKnownState:=TRUE,
    bMovingState:=FALSE,
    nPositionIndex:=1,
    stCurrentPosition:=astPositionState[1],
);
// Outside the deltas check
TestStaticPosition(
    nTestIndex:=1,
    sTestName:='OutsidePos1Delta',
    fPosition:=astPositionState[1].fPosition + 2 * astPositionState[1].fDelta,
    bKnownState:=FALSE,
    bMovingState:=FALSE,
    nPositionIndex:=0,
    stCurrentPosition:=stDummyPos,
);
// At invalid state 2 check
TestStaticPosition(
    nTestIndex:=2,
    sTestName:='AtInvalidPos',
    fPosition:=astPositionState[2].fPosition,
    bKnownState:=FALSE,
    bMovingState:=FALSE,
    nPositionIndex:=0,
    stCurrentPosition:=stDummyPos,
);
// At position 3 check
TestStaticPosition(
    nTestIndex:=3,
    sTestName:='AtPos3',
    fPosition:=astPositionState[3].fPosition - 0.5 * astPositionState[3].fDelta,
    bKnownState:=TRUE,
    bMovingState:=FALSE,
    nPositionIndex:=3,
    stCurrentPosition:=astPositionState[3],
);
// At position 3 and moving within bounds check
TestMovingPosition(
    nTestIndex:=4,
    sTestName:='MovingAt3',
    fStartPosition:=astPositionState[3].fPosition,
    fGoalPosition:=astPositionState[3].fPosition + 0.9 * astPositionState[3].fDelta,
    fVelocity:=0.001,
    bKnownState:=TRUE,
    bMovingState:=FALSE,
    nPositionIndex:=3,
    stCurrentPosition:=astPositionState[3],
);
// At position 3 and moving away check
TestMovingPosition(
    nTestIndex:=5,
    sTestName:='MovingFrom3',
    fStartPosition:=astPositionState[3].fPosition,
    fGoalPosition:=astPositionState[3].fPosition + 100 * astPositionState[3].fDelta,
    fVelocity:=0.001,
    bKnownState:=FALSE,
    bMovingState:=TRUE,
    nPositionIndex:=0,
    stCurrentPosition:=stDummyPos,
);
TestDupe(nTestIndex:=6);

IF bOneTestDone THEN
    bOneTestDone := FALSE;
    nTestCounter := nTestCounter + 1;
    fbTestMove(
        stMotionStage:=stMotionStage,
        bExecute:=FALSE,
    );
END_IF

METHOD PRIVATE Asserts
VAR_INPUT
    tTimeout: TIME;
    bKnownState: BOOL;
    bMovingState: BOOL;
    nPositionIndex: DINT;
    stCurrentPosition: ST_PositionState;
END_VAR
VAR
    abExpected: ARRAY[1..GeneralConstants.MAX_STATES] OF BOOL;
END_VAR

fbRead(
    stMotionStage:=stMotionStage,
    astPositionState:=astPositionstate,
);

AssertEquals_BOOL(
    Expected:=FALSE,
    Actual:=fbTestMove.tElapsed > tTimeout,
    Message:='Test timed out',
);
AssertEquals_BOOL(
    Expected:=bKnownState,
    Actual:=fbRead.bKnownState,
    Message:='Incorrect bKnownState',
);
AssertEquals_BOOL(
    Expected:=bMovingState,
    Actual:=fbRead.bMovingState,
    Message:='Incorrect bMovingState',
);
AssertEquals_DINT(
    Expected:=nPositionIndex,
    Actual:=fbRead.nPositionIndex,
    Message:='Incorrect nPositionIndex',
);
IF nPositionIndex > 0 THEN
    IF nPositionIndex <= GeneralConstants.MAX_STATES THEN
        abExpected[nPositionIndex] := TRUE;
    END_IF
 END_IF
AssertArrayEquals_BOOL(
    Expecteds:=abExpected,
    Actuals:=fbRead.abAtPosition,
    Message:='Wrong at position array',
);

IF bKnownState THEN
    AssertEquals_STRING(
        Expected:=stCurrentPosition.sName,
        Actual:=fbRead.stCurrentPosition.sName,
        Message:='Did not provide correct current position struct',
    );
END_IF
END_METHOD

METHOD TestDupe
VAR_INPUT
    nTestIndex: DINT;
END_VAR
VAR
    abExpected: ARRAY[1..GeneralConstants.MAX_STATES] OF BOOL;
END_VAR

TEST('TestDupe');
IF nTestIndex <> nTestCounter THEN
    RETURN;
END_IF

// In this test, and only in this test, we must make sure state 4 is valid
astPositionState[4].bValid := TRUE;

fbTestMove(
    stMotionStage:=stMotionStage,
    bExecute:=TRUE,
    fStartPosition:=astPositionState[4].fPosition,
    fGoalPosition:=astPositionState[4].fPosition,
);
abExpected[3] := TRUE;
abExpected[4] := TRUE;

IF fbTestMove.tElapsed > T#1s OR (fbTestMove.bSetDone AND bStatesReady) THEN
    fbRead(
        stMotionStage:=stMotionStage,
        astPositionState:=astPositionstate,
    );
    AssertEquals_BOOL(
        Expected:=FALSE,
        Actual:=fbTestMove.tElapsed > T#1s,
        Message:='Test timed out',
    );
    AssertEquals_BOOL(
        Expected:=TRUE,
        Actual:=fbRead.bKnownState,
        Message:='Incorrect bKnownState',
    );
    AssertArrayEquals_BOOL(
        Expecteds:=abExpected,
        Actuals:=fbRead.abAtPosition,
        Message:='Wrong at position array',
    );
    bOneTestDone := TRUE;
    TEST_FINISHED();
END_IF
END_METHOD

METHOD PRIVATE TestMovingPosition
VAR_INPUT
    nTestIndex: UINT;
    sTestName: STRING;
    fStartPosition: LREAL;
    fGoalPosition: LREAL;
    fVelocity: LREAL;
    bKnownState: BOOL;
    bMovingState: BOOL;
    nPositionIndex: DINT;
    stCurrentPosition: ST_PositionState;
END_VAR

TEST(sTestName);
IF nTestIndex <> nTestCounter THEN
    RETURN;
END_IF

fbTestMove(
    stMotionStage:=stMotionStage,
    bExecute:=TRUE,
    fStartPosition:=fStartPosition,
    fGoalPosition:=fGoalPosition,
    fVelocity:=0.001,
    bHWEnable:=TRUE,
);

IF fbTestMove.tElapsed > T#5s OR (fbTestMove.bMotionStarted AND bStatesReady) THEN
    Asserts(
        tTimeout:=T#5s,
        bKnownState:=bKnownState,
        bMovingState:=bMovingState,
        nPositionIndex:=nPositionIndex,
        stCurrentPosition:=stCurrentPosition,
    );
    bOneTestDone := TRUE;
    TEST_FINISHED();
END_IF
END_METHOD

METHOD PRIVATE TestStaticPosition
VAR_INPUT
    nTestIndex: UINT;
    sTestName: STRING;
    fPosition: LREAL;
    bKnownState: BOOL;
    bMovingState: BOOL;
    nPositionIndex: DINT;
    stCurrentPosition: ST_PositionState;
END_VAR

TEST(sTestName);
IF nTestIndex <> nTestCounter THEN
    RETURN;
END_IF

fbTestMove(
    stMotionStage:=stMotionStage,
    bExecute:=TRUE,
    fStartPosition:=fPosition,
    fGoalPosition:=fPosition,
);

IF fbTestMove.tElapsed > T#1s OR (fbTestMove.bSetDone AND bStatesReady) THEN
    Asserts(
        tTimeout:=T#1s,
        bKnownState:=bKnownState,
        bMovingState:=bMovingState,
        nPositionIndex:=nPositionIndex,
        stCurrentPosition:=stCurrentPosition,
    );
    bOneTestDone := TRUE;
    TEST_FINISHED();
END_IF
END_METHOD

END_FUNCTION_BLOCK

// Tests/FB_PositionStateReadND_Test
FUNCTION_BLOCK FB_PositionStateReadND_Test EXTENDS FB_MotorTestSuite
(*
    Test that FB_PositionStateReadND can be used to read and summarize
    N-dimensional state positions where multiple motors must move in
    sync to a shared named state.
*)
VAR
    astMotionStage: ARRAY[1..MotionConstants.MAX_STATE_MOTORS] OF ST_MotionStage;
    afbMotionStage: ARRAY[1..3] OF FB_MotionStage;
    astPositionState: ARRAY[1..MotionConstants.MAX_STATE_MOTORS] OF ARRAY [1..GeneralConstants.MAX_STATES] OF ST_PositionState;
    afbInternal: ARRAY[1..3] OF ARRAY [1..2] OF FB_PositionStateInternal;

    afbTestMove: ARRAY[1..3] OF FB_TestHelperSetAndMove;
    fbRead: FB_PositionStateReadND;
    bOneAssertDone: BOOL;
    nAssertCounter: UINT;
    nIter1: UINT;
    nIter2: UINT;
    nIter3: UINT;

    fbMisRead: FB_PositionStateReadND;
    astGoodStage: ARRAY[1..MotionConstants.MAX_STATE_MOTORS] OF ST_MotionStage;
    astGoodStateShape: ARRAY[1..MotionConstants.MAX_STATE_MOTORS] OF ARRAY [1..GeneralConstants.MAX_STATES] OF ST_PositionState;

    astSqMotionStage: ARRAY[1..MotionConstants.MAX_STATE_MOTORS] OF ST_MotionStage;
    afbSqMotionStage: ARRAY[1..2] OF FB_MotionStage;
    astSquareStates: ARRAY[1..MotionConstants.MAX_STATE_MOTORS] OF ARRAY [1..GeneralConstants.MAX_STATES] OF ST_PositionState;
    afbSqInternal: ARRAY[1..2] OF ARRAY[1..4] OF FB_PositionStateInternal;

    afbSqTestMove: ARRAY[1..2] OF FB_TestHelperSetAndMove;
    fbSqRead: FB_PositionStateReadND;
    bSqAssertDone: BOOL;
    nSqAssertCounter: UINT;
END_VAR
VAR CONSTANT
    NO_STATE: UINT := 0;
    OUT_STATE: UINT := 1;
    IN_STATE: UINT := 2;
    IN_TWEAK: UINT := 3;
    AWAY: UINT := 4;
    LAST_TEST: UINT := AWAY;
    TEST_COUNT: UINT := 5;
END_VAR


PerMotor(1);
PerMotor(2);
PerMotor(3);
SquareSetup();

// First check the case of mismatched arrays
TestForgot();
TestCombos(nAssertCounter);
TestSquare(nSqAssertCounter);

IF bOneAssertDone THEN
    afbTestMove[1](
        stMotionStage:=astMotionStage[1],
        bExecute:=FALSE,
    );
    afbTestMove[2](
        stMotionStage:=astMotionStage[2],
        bExecute:=FALSE,
    );
    afbTestMove[3](
        stMotionStage:=astMotionStage[3],
        bExecute:=FALSE,
    );
    IF afbTestMove[1].bResetDone AND afbTestMove[2].bResetDone AND afbTestMove[3].bResetDone THEN
        bOneAssertDone := FALSE;
        nAssertCounter := nAssertCounter + 1;
    END_IF
END_IF

IF bSqAssertDone THEN
    afbSqTestMove[1](
        stMotionStage:=astMotionStage[1],
        bExecute:=FALSE,
    );
    afbSqTestMove[2](
        stMotionStage:=astMotionStage[2],
        bExecute:=FALSE,
    );
    IF afbSqTestMove[1].bResetDone AND afbSqTestMove[2].bResetDone THEN
        bSqAssertDone := FALSE;
        nSqAssertCounter := nSqAssertCounter + 1;
    END_IF
END_IF

METHOD PRIVATE DoAssert
VAR_INPUT
    nMotorCase1: UINT;
    nMotorCase2: UINT;
    nMotorCase3: UINT;
    bReady1: BOOL;
    bReady2: BOOL;
    bReady3: BOOL;
END_VAR
VAR
    bKnownState: BOOL;
    bMovingState: BOOL;
    nPositionIndex: DINT;
    sTestCase: STRING;
END_VAR

sTestCase := CONCAT(CONCAT(UINT_TO_STRING(nMotorCase1), UINT_TO_STRING(nMotorCase2)), UINT_TO_STRING(nMotorCase3));

AssertTrue(
    Condition:=bReady1,
    Message:=CONCAT('Timeout for motor 1 during test case ', sTestCase),
);
AssertTrue(
    Condition:=bReady2,
    Message:=CONCAT('Timeout for motor 2 during test case ', sTestCase),
);
AssertTrue(
    Condition:=bReady3,
    Message:=CONCAT('Timeout for motor 3 during test case ', sTestCase),
);

// All at OUT or all at IN should be OUT and IN respectively, even if doing a tweak move
// Any other combination is at no state
IF nMotorCase1 = OUT_STATE AND nMotorCase2 = OUT_STATE AND nMotorCase3 = OUT_STATE THEN
    bKnownState := TRUE;
    nPositionIndex := 1;
ELSIF (nMotorCase1 = IN_STATE OR nMotorCase1 = IN_TWEAK) AND
      (nMotorCase2 = IN_STATE OR nMotorCase2 = IN_TWEAK) AND
      (nMotorCase3 = IN_STATE OR nMotorCase3 = IN_TWEAK) THEN
    bKnownState := TRUE;
    nPositionIndex := 2;
END_IF
// In addition, bMovingState must be set if any is moving away from a state
IF nMotorCase1 = AWAY OR nMotorCase2 = AWAY OR nMotorCase3 = AWAY THEN
    bMovingState := TRUE;
END_IF

AssertEquals_BOOL(
    Expected:=bKnownState,
    Actual:=fbRead.bKnownState,
    Message:=CONCAT('Wrong bKnownState for test case ', sTestCase),
);
AssertEquals_BOOL(
    Expected:=bMovingState,
    Actual:=fbRead.bMovingState,
    Message:=CONCAT('Wrong bMovingState for test case ', sTestCase),
);
AssertEquals_DINT(
    Expected:=nPositionIndex,
    Actual:=fbRead.nPositionIndex,
    Message:=CONCAT('Wrong nPositionIndex for test case ', sTestCase),
);
END_METHOD

METHOD PRIVATE DoMove: BOOL
VAR_INPUT
    nMotorIndex: UINT;
    nMotorCase: UINT;
END_VAR
VAR
    fStartPosition: LREAL;
    fGoalPosition: LREAL;
END_VAR

CASE nMotorCase OF
    // Somewhere smaller than OUT, static
    NO_STATE:
        fStartPosition := astPositionState[nMotorIndex][1].fPosition - 10 * astPositionState[nMotorIndex][1].fDelta;
        fGoalPosition := fStartPosition;
    // Exactly at OUT, static
    OUT_STATE:
        fStartPosition := astPositionState[nMotorIndex][1].fPosition;
        fGoalPosition := fStartPosition;
    // Exactly at IN, static
    IN_STATE:
        fStartPosition := astPositionState[nMotorIndex][2].fPosition;
        fGoalPosition := fStartPosition;
    // Start at IN, do a small tweak
    IN_TWEAK:
        fStartPosition := astPositionState[nMotorIndex][2].fPosition;
        fGoalPosition := fStartPosition + 0.9 * astPositionState[nMotorIndex][2].fDelta;
    // Start at IN, move positive a lot
    AWAY:
        fStartPosition := astPositionState[nMotorIndex][2].fPosition;
        fGoalPosition := fStartPosition + 100 * astPositionState[nMotorIndex][2].fDelta;
END_CASE

afbTestMove[nMotorIndex](
    stMotionStage:=astMotionStage[nMotorIndex],
    bExecute:=TRUE,
    fStartPosition:=fStartPosition,
    fGoalPosition:=fGoalPosition,
    fVelocity:=0.001,
    bHWEnable:=TRUE,
);

CASE nMotorCase OF
    // All static states: report ready when set is done
    NO_STATE:
        DoMove := afbTestMove[nMotorIndex].bSetDone;
    OUT_STATE:
        DoMove := afbTestMove[nMotorIndex].bSetDone;
    IN_STATE:
        DoMove := afbTestMove[nMotorIndex].bSetDone;
    // All moving states: report ready when move starts
    IN_TWEAK:
        DoMove := afbTestMove[nMotorIndex].bMotionStarted;
    AWAY:
        DoMove := afbTestMove[nMotorIndex].bMotionStarted;
END_CASE
// Universal 5s timeout
DoMove S= afbTestMove[nMotorIndex].tElapsed > T#5s;
END_METHOD

METHOD PRIVATE DoRead
VAR_INPUT
END_VAR

fbRead(
    astMotionStage:=astMotionStage,
    astPositionState:=astPositionState,
    nActiveMotorCount:=3,
);
END_METHOD

METHOD PRIVATE PerMotor : BOOL
VAR_INPUT
    nIndex: DINT;
END_VAR

afbMotionStage[nIndex](stMotionStage:=astMotionStage[nIndex]);

astPositionState[nIndex][1].sName := 'OUT';
astPositionState[nIndex][1].fPosition := nIndex * 100 + 10;
astPositionState[nIndex][1].fDelta := 1;
astPositionState[nIndex][1].bUseRawCounts := FALSE;
SetGoodState(astPositionState[nIndex][1]);
afbInternal[nIndex][1](
    stMotionStage:=astMotionStage[nIndex],
    stPositionState:=astPositionState[nIndex][1],
);

astPositionState[nIndex][2].sName := 'IN';
astPositionState[nIndex][2].fPosition := nIndex * 100 + 20;
astPositionState[nIndex][2].fDelta := 1;
astPositionState[nIndex][2].bUseRawCounts := FALSE;
SetGoodState(astPositionState[nIndex][2]);
afbInternal[nIndex][2](
    stMotionStage:=astMotionStage[nIndex],
    stPositionState:=astPositionState[nIndex][2],
);
END_METHOD

METHOD SquareSetup
VAR_INPUT
END_VAR
// 2 motors, 4 positions per motor, square geometry
// Motor 1 is X, motor 2 is Y
// Corners at (10,10), (10, 20), (20, 10), (20, 20)
// So motor 1 is either LEFT=10 or RIGHT=20
// motor 2 is either BOT=10 or TOP=20

afbSqMotionStage[1](stMotionStage:=astSqMotionStage[1]);
afbSqMotionStage[2](stMotionStage:=astSqMotionStage[2]);

astSquareStates[1][1].sName := 'Top Left';
astSquareStates[1][1].fPosition := 10;
astSquareStates[1][1].fDelta := 1;
SetGoodState(astSquareStates[1][1]);
afbSqInternal[1][1](
    stMotionStage:=astMotionStage[1],
    stPositionState:=astSquareStates[1][1],
);

astSquareStates[1][2].sName := 'Top Right';
astSquareStates[1][2].fPosition := 20;
astSquareStates[1][2].fDelta := 1;
SetGoodState(astSquareStates[1][2]);
afbSqInternal[1][2](
    stMotionStage:=astMotionStage[1],
    stPositionState:=astSquareStates[1][2],
);

astSquareStates[1][3].sName := 'Bot Left';
astSquareStates[1][3].fPosition := 10;
astSquareStates[1][3].fDelta := 1;
SetGoodState(astSquareStates[1][3]);
afbSqInternal[1][3](
    stMotionStage:=astMotionStage[1],
    stPositionState:=astSquareStates[1][3],
);

astSquareStates[1][4].sName := 'Bot Right';
astSquareStates[1][4].fPosition := 20;
astSquareStates[1][4].fDelta := 1;
SetGoodState(astSquareStates[1][4]);
afbSqInternal[1][4](
    stMotionStage:=astMotionStage[1],
    stPositionState:=astSquareStates[1][4],
);

astSquareStates[2][1].sName := 'Top Left';
astSquareStates[2][1].fPosition := 20;
astSquareStates[2][1].fDelta := 1;
SetGoodState(astSquareStates[2][1]);
afbSqInternal[2][1](
    stMotionStage:=astMotionStage[1],
    stPositionState:=astSquareStates[2][1],
);

astSquareStates[2][2].sName := 'Top Right';
astSquareStates[2][2].fPosition := 20;
astSquareStates[2][2].fDelta := 1;
SetGoodState(astSquareStates[2][2]);
afbSqInternal[2][2](
    stMotionStage:=astMotionStage[1],
    stPositionState:=astSquareStates[2][2],
);

astSquareStates[2][3].sName := 'Bot Left';
astSquareStates[2][3].fPosition := 10;
astSquareStates[2][3].fDelta := 1;
SetGoodState(astSquareStates[2][3]);
afbSqInternal[2][3](
    stMotionStage:=astMotionStage[1],
    stPositionState:=astSquareStates[2][3],
);

astSquareStates[2][4].sName := 'Bot Right';
astSquareStates[2][4].fPosition := 10;
astSquareStates[2][4].fDelta := 1;
SetGoodState(astSquareStates[2][4]);
afbSqInternal[2][4](
    stMotionStage:=astMotionStage[1],
    stPositionState:=astSquareStates[2][4],
);
END_METHOD

METHOD PRIVATE TestCombos
VAR_INPUT
    nAssertID: UINT;
END_VAR
VAR
    nMotor1Case: UINT;
    nMotor2Case: UINT;
    nMotor3Case: UINT;
    bReady1: BOOL;
    bReady2: BOOL;
    bReady3: BOOL;
END_VAR
VAR_INST
    tonTimeout: TON;
END_VAR

// This should be one big test case with 125 asserts
TEST('TestAllCombos');

nMotor1Case := nAssertID MOD TEST_COUNT;
nMotor2Case := LREAL_TO_UINT(FLOOR(nAssertID / TEST_COUNT)) MOD TEST_COUNT;
nMotor3Case := LREAL_TO_UINT(FLOOR(nAssertID / TEST_COUNT / TEST_COUNT)) MOD TEST_COUNT;

bReady1 := DoMove(1, nMotor1Case);
bReady2 := DoMove(2, nMotor2Case);
bReady3 := DoMove(3, nMotor3Case);

// There is a 5s timeout at a lower level, but that timeout could fail
tonTimeout(
    IN:=TRUE,
    PT:=T#7s,
);

IF tonTimeout.Q OR (bReady1 AND bReady2 AND bReady3) THEN
    DoRead();
    DoAssert(nMotor1Case, nMotor2Case, nMotor3Case, bReady1, bReady2, bReady3);
    bOneAssertDone := TRUE;
    // The final assert case marks test as finished
    IF tonTimeout.Q OR (nMotor1Case = LAST_TEST AND nMotor2Case = LAST_TEST AND nMotor3Case = LAST_TEST) THEN
        // 11 extra tests
        // 1 from TestForgot
        // 10 (2*5) from TestSquare
        AssertEquals_UINT(
            Expected:=6 * TEST_COUNT * TEST_COUNT * TEST_COUNT + 11,
            Actual:=AssertResults.TotalAsserts,
            Message:='Some of the asserts were not run',
        );
        AssertFalse(
            tonTimeout.Q,
            'Level 2 timeout in test',
        );
        TEST_FINISHED();
    END_IF
    tonTimeout(IN:=FALSE);
END_IF
END_METHOD

METHOD PRIVATE TestForgot
VAR
END_VAR

TEST('ForgotCount');

fbMisRead(
    astMotionStage:=astGoodStage,
    astPositionState:=astGoodStateShape,
);

AssertTrue(
    Condition:=fbMisRead.bMotorCountError,
    Message:='Failed to notice missing count',
);

TEST_FINISHED();
END_METHOD

METHOD TestSquare
VAR_INPUT
    nAssertID: UINT;
END_VAR
VAR
    fMotor1Pos: LREAL;
    fMotor2Pos: LREAL;
    nGoal: UINT;
END_VAR
VAR_INST
    tonTimeout: TON;
END_VAR

// We'll do 5 tests, one at each square point and one more in the middle
Test('TestSquare');
IF nAssertID > 4 THEN
    RETURN;
END_IF

IF nAssertID = 0 THEN
    fMotor1Pos := 10;
    fMotor2Pos := 10;
    nGoal := 3;
ELSIF nAssertID = 1 THEN
    fMotor1Pos := 20;
    fMotor2Pos := 10;
    nGoal := 4;
ELSIF nAssertID = 2 THEN
    fMotor1Pos := 10;
    fMotor2Pos := 20;
    nGoal := 1;
ELSIF nAssertID = 3 THEN
    fMotor1Pos := 20;
    fMotor2Pos := 20;
    nGoal := 2;
ELSIF nAssertID = 4 THEN
    fMotor1Pos := 15;
    fMotor2Pos := 15;
    nGoal := 0;
END_IF

afbSqTestMove[1](
    stMotionStage:=astSqMotionStage[1],
    bExecute:=TRUE,
    fStartPosition:=fMotor1Pos,
    fGoalPosition:=fMotor1Pos,
);
afbSqTestMove[2](
    stMotionStage:=astSqMotionStage[2],
    bExecute:=TRUE,
    fStartPosition:=fMotor2Pos,
    fGoalPosition:=fMotor2Pos,
);

tonTimeout(
    IN:=TRUE,
    PT:=T#5s,
);

IF tonTimeout.Q OR afbSqTestMove[1].bSetDone AND afbSqTestMove[1].bSetDone THEN
    fbSqRead(
        astMotionStage:=astSqMotionStage,
        astPositionState:=astSquareStates,
        nActiveMotorCount:=2,
    );
    AssertFalse(
        tonTimeout.Q,
        CONCAT('Timeout in square test ', UINT_TO_STRING(nAssertID)),
    );
    AssertEquals_UINT(
        Expected:=nGoal,
        Actual:=fbSqRead.nPositionIndex,
        Message:=CONCAT('Wrong read in square test ', UINT_TO_STRING(nAssertID)),
    );

    bSqAssertDone := TRUE;
    IF nAssertID = 4 THEN
        TEST_FINISHED();
    END_IF
    tonTimeout(IN:=FALSE);
END_IF
END_METHOD

END_FUNCTION_BLOCK

// Tests/FB_StatePMPSEnables_Test
FUNCTION_BLOCK FB_StatePMPSEnables_Test EXTENDS FB_MotorTestSuite
(*
    Tests for FB_StatePMPSEnables

    This function block ensures that:
    - When not at our goal state, we cannot move away from our goal state
    - When at our goal state, we must stay within the state bounds
    - When at our goal state, we still obey other constraints like limit switches

    We also include a super basic real move test with our simulator motor to make sure the enables are set properly.
*)
VAR
    stMotionStage: ST_MotionStage;
    fbMotionStage: FB_MotionStage;
    astPositionState: ARRAY[1..GeneralConstants.MAX_STATES] OF ST_PositionState;
    fbInternal1: FB_PositionStateInternal;
    fbInternal2: FB_PositionStateInternal;
    nInvalidState: UINT := 2;
    nGoalState: UINT := 4;
    nNotUpdatedState: UINT := 6;

    bInit: BOOL;
    nTestCounter: UINT;
    bOneTestDone: BOOL;
    fTestStartPos: LREAL;
    tonTimer: TON;
    bStatesReady: BOOL;
END_VAR


astPositionState[nGoalState].fPosition := 10;
astPositionState[nGoalState].fDelta := 1;
SetGoodState(astPositionState[nGoalState]);
astPositionState[nInvalidState].fPosition := 20;
astPositionState[nInvalidState].fDelta := 1;
astPositionState[nNotUpdatedState].fPosition := 20;
astPositionState[nNotUpdatedState].fDelta := 1;
SetGoodState(astPositionState[nNotUpdatedState]);
fbInternal1(
    stMotionStage:=stMotionStage,
    stPositionState:=astPositionState[nGoalState],
);
fbInternal2(
    stMotionStage:=stMotionStage,
    stPositionState:=astPositionState[nInvalidState],
);
fbMotionStage(stMotionStage:=stMotionStage);
bStatesReady:=astPositionState[nGoalState].bUpdated AND astPositionState[nInvalidState].bUpdated;

IF bStatesReady AND nTestCounter = 0 THEN
    // Don't run any tests until the states are ready
    nTestCounter := 1;
END_IF

TestInvalid(1);
TestNotUpdated(2);
TestBelow(3);
TestAbove(4);
TestAt(5);
TestDisabled(6);
TestLimits(7);
TestMoveTo(8);
TestMoveAt(9);

IF bOneTestDone THEN
    bOneTestDone := FALSE;
    nTestCounter := nTestCounter + 1;
    tonTimer(IN:=FALSE);
END_IF
// Use this timer to time out any tests that stall
tonTimer(
    IN:=bStatesReady,
    PT:=T#5s,
);

METHOD TestAbove
VAR_INPUT
    nTestID: UINT;
END_VAR
VAR_INST
    fbStateEnables: FB_StatePMPSEnables;
    fbFFHWO: FB_HardwareFFOutput := (bAutoReset := TRUE);
    fbMove: FB_TestHelperSetAndMove;

    bInit: BOOL;
END_VAR

TEST('TestAbove');
IF nTestCounter <> nTestID THEN
    RETURN;
END_IF

SetEnablesPMPS(stMotionStage);

// Set position to be above the goal's range
fbMove(
    stMotionStage:=stMotionStage,
    bExecute:=bInit,
    fStartPosition:=astPositionState[nGoalState].fPosition + 100 * astPositionState[nGoalState].fDelta,
    fGoalPosition:=astPositionState[nGoalState].fPosition + 100 * astPositionState[nGoalState].fDelta,
    fVelocity:=1,
    bHWEnable:=FALSE,
);
bInit := TRUE;
// Run our FB
fbStateEnables(
    stMotionStage:=stMotionStage,
    astPositionState:=astPositionState,
    fbFFHWO:=fbFFHWO,
    bEnable:=TRUE,
    nGoalStateIndex:=nGoalState,
);
fbFFHWO.EvaluateOutput();
// If we've set the position OR ran out of time to set the position, check the asserts
IF tonTimer.Q OR fbMove.bSetDone THEN
    AssertFalse(
        tonTimer.Q,
        'Timeout in test',
    );
    AssertEquals_LREAL(
        Expected:=fbMove.fStartPosition,
        Actual:=fbMove.fActPosition,
        Delta:=0.0001,
        Message:='Position was not set correctly',
    );
    AssertTrue(
        fbFFHWO.q_xFastFaultOut,
        'Fast fault in normal situation',
    );
    AssertFalse(
        fbStateEnables.bForwardEnabled,
        'Forward enabled when above goal',
    );
    AssertTrue(
        fbStateEnables.bBackwardEnabled,
        'Backward disabled when above goal',
    );
    bOneTestDone := TRUE;
    TEST_FINISHED();
END_IF
END_METHOD

METHOD TestAt
VAR_INPUT
    nTestID: UINT;
END_VAR
VAR_INST
    fbStateEnables: FB_StatePMPSEnables;
    fbFFHWO: FB_HardwareFFOutput := (bAutoReset := TRUE);
    fbMove: FB_TestHelperSetAndMove;

    bInit: BOOL;
END_VAR

TEST('TestAt');
IF nTestCounter <> nTestID THEN
    RETURN;
END_IF

SetEnablesPMPS(stMotionStage);

// Set position to be at the goal state
fbMove(
    stMotionStage:=stMotionStage,
    bExecute:=bInit,
    fStartPosition:=astPositionState[nGoalState].fPosition,
    fGoalPosition:=astPositionState[nGoalState].fPosition,
    fVelocity:=1,
    bHWEnable:=FALSE,
);
bInit := TRUE;
// Run our FB
fbStateEnables(
    stMotionStage:=stMotionStage,
    astPositionState:=astPositionState,
    fbFFHWO:=fbFFHWO,
    bEnable:=TRUE,
    nGoalStateIndex:=nGoalState,
);
fbFFHWO.EvaluateOutput();
// If we've set the position OR ran out of time to set the position, check the asserts
IF tonTimer.Q OR fbMove.bSetDone THEN
    AssertFalse(
        tonTimer.Q,
        'Timeout in test',
    );
    AssertEquals_LREAL(
        Expected:=fbMove.fStartPosition,
        Actual:=fbMove.fActPosition,
        Delta:=0.0001,
        Message:='Position was not set correctly',
    );
    AssertTrue(
        fbFFHWO.q_xFastFaultOut,
        'Fast fault in normal situation',
    );
    AssertTrue(
        fbStateEnables.bForwardEnabled,
        'Forward disabled when at goal',
    );
    AssertTrue(
        fbStateEnables.bBackwardEnabled,
        'Backward disabled when at goal',
    );
    bOneTestDone := TRUE;
    TEST_FINISHED();
END_IF
END_METHOD

METHOD TestBelow
VAR_INPUT
    nTestID: UINT;
END_VAR
VAR_INST
    fbStateEnables: FB_StatePMPSEnables;
    fbFFHWO: FB_HardwareFFOutput := (bAutoReset := TRUE);
    fbMove: FB_TestHelperSetAndMove;

    bInit: BOOL;
END_VAR

TEST('TestBelow');
IF nTestCounter <> nTestID THEN
    RETURN;
END_IF

SetEnablesPMPS(stMotionStage);

// Set position to be below the goal's range
fbMove(
    stMotionStage:=stMotionStage,
    bExecute:=bInit,
    fStartPosition:=astPositionState[nGoalState].fPosition - 100 * astPositionState[nGoalState].fDelta,
    fGoalPosition:=astPositionState[nGoalState].fPosition - 100 * astPositionState[nGoalState].fDelta,
    fVelocity:=1,
    bHWEnable:=FALSE,
);
bInit := TRUE;
// Run our FB
fbStateEnables(
    stMotionStage:=stMotionStage,
    astPositionState:=astPositionState,
    fbFFHWO:=fbFFHWO,
    bEnable:=bInit,
    nGoalStateIndex:=nGoalState,
);

fbFFHWO.EvaluateOutput();
// If we've set the position OR ran out of time to set the position, check the asserts
IF tonTimer.Q OR fbMove.bSetDone THEN
    AssertFalse(
        tonTimer.Q,
        'Timeout in test',
    );
    AssertEquals_LREAL(
        Expected:=fbMove.fStartPosition,
        Actual:=fbMove.fActPosition,
        Delta:=0.0001,
        Message:='Position was not set correctly',
    );
    AssertTrue(
        fbFFHWO.q_xFastFaultOut,
        'Fast fault in normal situation',
    );
    AssertFalse(
        fbStateEnables.bBackwardEnabled,
        'Backward enabled when below goal',
    );
    AssertTrue(
        fbStateEnables.bForwardEnabled,
        'Forward disabled when below goal',
    );
    bOneTestDone := TRUE;
    TEST_FINISHED();
END_IF
END_METHOD

METHOD TestDisabled
VAR_INPUT
    nTestID: UINT;
END_VAR
VAR_INST
    fbStateEnables: FB_StatePMPSEnables;
    fbFFHWO: FB_HardwareFFOutput := (bAutoReset := TRUE);
    fbMove: FB_TestHelperSetAndMove;

    bInit: BOOL;
END_VAR

TEST('TestDisabled');
IF nTestCounter <> nTestID THEN
    RETURN;
END_IF

SetEnablesPMPS(stMotionStage);

// Set position to be below the goal's range
fbMove(
    stMotionStage:=stMotionStage,
    bExecute:=bInit,
    fStartPosition:=astPositionState[nGoalState].fPosition - 100 * astPositionState[nGoalState].fDelta,
    fGoalPosition:=astPositionState[nGoalState].fPosition - 100 * astPositionState[nGoalState].fDelta,
    fVelocity:=1,
    bHWEnable:=FALSE,
);
bInit := TRUE;
// Run our FB
fbStateEnables(
    stMotionStage:=stMotionStage,
    astPositionState:=astPositionState,
    fbFFHWO:=fbFFHWO,
    bEnable:=FALSE,
    nGoalStateIndex:=nGoalState,
);

fbFFHWO.EvaluateOutput();
// If we've set the position OR ran out of time to set the position, check the asserts
IF tonTimer.Q OR fbMove.bSetDone THEN
    AssertFalse(
        tonTimer.Q,
        'Timeout in test',
    );
    AssertEquals_LREAL(
        Expected:=fbMove.fStartPosition,
        Actual:=fbMove.fActPosition,
        Delta:=0.0001,
        Message:='Position was not set correctly',
    );
    AssertTrue(
        fbFFHWO.q_xFastFaultOut,
        'Fast fault in normal situation',
    );
    AssertTrue(
        fbStateEnables.bBackwardEnabled,
        'Backward disabled when fb is supposed to be disabled',
    );
    AssertTrue(
        fbStateEnables.bForwardEnabled,
        'Forward disabled when fb is supposed to be disabled',
    );
    bOneTestDone := TRUE;
    TEST_FINISHED();
END_IF
END_METHOD

METHOD TestInvalid
VAR_INPUT
    nTestID: UINT;
END_VAR
VAR_INST
    fbStateEnables: FB_StatePMPSEnables;
    fbFFHWO: FB_HardwareFFOutput := (bAutoReset := TRUE);
END_VAR

TEST('TestInvalid');
IF nTestCounter <> nTestID THEN
    RETURN;
END_IF

SetEnablesPMPS(stMotionStage);

fbFFHWO.EvaluateOutput();
AssertTrue(
    fbFFHWO.q_xFastFaultOut,
    'Faulted prior to test',
);
// The invalid state should give us a fault
fbStateEnables(
    stMotionStage:=stMotionStage,
    astPositionState:=astPositionState,
    fbFFHWO:=fbFFHWO,
    bEnable:=TRUE,
    nGoalStateIndex:=nInvalidState,
);
fbFFHWO.EvaluateOutput();
AssertFalse(
    fbFFHWO.q_xFastFaultOut,
    'Invalid state did not fault',
);

bOneTestDone := TRUE;
TEST_FINISHED();
END_METHOD

METHOD TestLimits
VAR_INPUT
    nTestID: UINT;
END_VAR
VAR_INST
    fbStateEnables: FB_StatePMPSEnables;
    fbFFHWO: FB_HardwareFFOutput := (bAutoReset := TRUE);
    fbMove: FB_TestHelperSetAndMove;

    bInit: BOOL;
END_VAR

TEST('TestLimits');
IF nTestCounter <> nTestID THEN
    RETURN;
END_IF

SetEnablesPMPS(stMotionStage);
// Kill the limit switches for this test
stMotionStage.bLimitForwardEnable := FALSE;
stMotionStage.bLimitBackwardEnable := FALSE;

// Set position to be at the goal state
fbMove(
    stMotionStage:=stMotionStage,
    bExecute:=bInit,
    fStartPosition:=astPositionState[nGoalState].fPosition,
    fGoalPosition:=astPositionState[nGoalState].fPosition,
    fVelocity:=1,
    bHWEnable:=FALSE,
);
bInit := TRUE;

// Run our FB
fbStateEnables(
    stMotionStage:=stMotionStage,
    astPositionState:=astPositionState,
    fbFFHWO:=fbFFHWO,
    bEnable:=TRUE,
    nGoalStateIndex:=nGoalState,
);
fbFFHWO.EvaluateOutput();
// If we've set the position OR ran out of time to set the position, check the asserts
IF tonTimer.Q OR fbMove.bSetDone THEN
    AssertFalse(
        tonTimer.Q,
        'Timeout in test',
    );
    AssertEquals_LREAL(
        Expected:=fbMove.fStartPosition,
        Actual:=fbMove.fActPosition,
        Delta:=0.0001,
        Message:='Position was not set correctly',
    );
    AssertTrue(
        fbFFHWO.q_xFastFaultOut,
        'Fast fault in normal situation',
    );
    AssertFalse(
        fbStateEnables.bForwardEnabled,
        'Forward enabled with limit hit',
    );
    AssertFalse(
        fbStateEnables.bBackwardEnabled,
        'Backward enabled with limit hit',
    );
    bOneTestDone := TRUE;
    TEST_FINISHED();
END_IF
END_METHOD

METHOD TestMoveAt
VAR_INPUT
    nTestID: UINT;
END_VAR
VAR_INST
    fbStateEnables: FB_StatePMPSEnables;
    fbFFHWO: FB_HardwareFFOutput := (bAutoReset := TRUE);
    fbMove: FB_TestHelperSetAndMove;

    bInit: BOOL;
END_VAR

TEST('TestMoveAt');
IF nTestCounter <> nTestID THEN
    RETURN;
END_IF

SetEnablesPMPS(stMotionStage);

// Run our FB which should enable the real move
fbStateEnables(
    stMotionStage:=stMotionStage,
    astPositionState:=astPositionState,
    fbFFHWO:=fbFFHWO,
    bEnable:=bInit,
    nGoalStateIndex:=nGoalState,
    eStatePMPSStatus:=E_StatePMPSStatus.AT_STATE,
    bTransitionAuthorized:=FALSE,
);

// Set position to be below the goal's range, and move to the goal
fbMove(
    stMotionStage:=stMotionStage,
    bExecute:=bInit,
    fStartPosition:=astPositionState[nGoalState].fPosition - astPositionState[nGoalState].fDelta / 2,
    fGoalPosition:=astPositionState[nGoalState].fPosition + astPositionState[nGoalState].fDelta / 2,
    fVelocity:=5,
    bHWEnable:=FALSE,
);
bInit := TRUE;

fbFFHWO.EvaluateOutput();

// If we've reached the position OR ran out of time to set the position, check the asserts
IF tonTimer.Q OR fbMove.bMoveDone THEN
    AssertFalse(
        tonTimer.Q,
        'Timeout in test',
    );
    AssertEquals_LREAL(
        Expected:=astPositionState[nGoalState].fPosition + astPositionState[nGoalState].fDelta / 2,
        Actual:=fbMove.fActPosition,
        Delta:=0.0001,
        Message:='Did not reach the goal position',
    );
    AssertTrue(
        fbFFHWO.q_xFastFaultOut,
        'Fast fault in normal situation',
    );
    AssertTrue(
        fbStateEnables.bBackwardEnabled,
        'Backward disabled when at goal',
    );
    AssertTrue(
        fbStateEnables.bForwardEnabled,
        'Forward disabled when at goal',
    );
    bOneTestDone := TRUE;
    TEST_FINISHED();
END_IF
END_METHOD

METHOD TestMoveTo
VAR_INPUT
    nTestID: UINT;
END_VAR
VAR_INST
    fbStateEnables: FB_StatePMPSEnables;
    fbFFHWO: FB_HardwareFFOutput := (bAutoReset := TRUE);
    fbMove: FB_TestHelperSetAndMove;

    bInit: BOOL;
END_VAR

TEST('TestMoveTo');
IF nTestCounter <> nTestID THEN
    RETURN;
END_IF

SetEnablesPMPS(stMotionStage);

// Run our FB which should enable the real move
fbStateEnables(
    stMotionStage:=stMotionStage,
    astPositionState:=astPositionState,
    fbFFHWO:=fbFFHWO,
    bEnable:=bInit,
    nGoalStateIndex:=nGoalState,
    eStatePMPSStatus:=E_StatePMPSStatus.TRANSITION,
    bTransitionAuthorized:=TRUE,
);

// Set position to be below the goal's range, and move to the goal
fbMove(
    stMotionStage:=stMotionStage,
    bExecute:=bInit,
    fStartPosition:=astPositionState[nGoalState].fPosition - 10,
    fGoalPosition:=astPositionState[nGoalState].fPosition,
    fVelocity:=5,
    bHWEnable:=FALSE,
);
bInit := TRUE;

fbFFHWO.EvaluateOutput();

// If we've reached the position OR ran out of time to set the position, check the asserts
IF tonTimer.Q OR fbMove.bMoveDone THEN
    AssertFalse(
        tonTimer.Q,
        'Timeout in test',
    );
    AssertEquals_LREAL(
        Expected:=astPositionState[nGoalState].fPosition,
        Actual:=fbMove.fActPosition,
        Delta:=0.0001,
        Message:='Did not reach the goal position',
    );
    AssertTrue(
        fbFFHWO.q_xFastFaultOut,
        'Fast fault in normal situation',
    );
    AssertTrue(
        fbStateEnables.bBackwardEnabled,
        'Backward disabled when at goal',
    );
    AssertTrue(
        fbStateEnables.bForwardEnabled,
        'Forward disabled when at goal',
    );
    bOneTestDone := TRUE;
    TEST_FINISHED();
END_IF
END_METHOD

METHOD TestNotUpdated
VAR_INPUT
    nTestID: UINT;
END_VAR
VAR_INST
    fbStateEnables: FB_StatePMPSEnables;
    fbFFHWO: FB_HardwareFFOutput := (bAutoReset := TRUE);
END_VAR

TEST('TestNotUpdated');
IF nTestCounter <> nTestID THEN
    RETURN;
END_IF

SetEnablesPMPS(stMotionStage);

fbFFHWO.EvaluateOutput();
AssertTrue(
    fbFFHWO.q_xFastFaultOut,
    'Faulted prior to test',
);
// The invalid state should give us a fault
fbStateEnables(
    stMotionStage:=stMotionStage,
    astPositionState:=astPositionState,
    fbFFHWO:=fbFFHWO,
    bEnable:=TRUE,
    nGoalStateIndex:=nNotUpdatedState,
);
fbFFHWO.EvaluateOutput();
AssertFalse(
    fbFFHWO.q_xFastFaultOut,
    'Not updated state did not fault',
);

bOneTestDone := TRUE;
TEST_FINISHED();
END_METHOD

END_FUNCTION_BLOCK

// Tests/FB_StatePMPSEnablesND_Test
FUNCTION_BLOCK FB_StatePMPSEnablesND_Test EXTENDS FB_MotorTestSuite
(*
    Unit tests for FB_StatePMPSEnablesND
    I'm confident that FB_StatePMPSEnables was tested in FB_StatePMPSEnables_Test
    There will be one core functionality check
    Then, the rest will be about the ND feature adds.
    Full checks:
    - Core motors not at goal can't move away check
    - bMaintMode = no move restrictions for all motors.
    - bMaintMode = fast fault
    - Wrong count = fast fault
*)
VAR
    astMotionStage: ARRAY[1..MotionConstants.MAX_STATE_MOTORS] OF ST_MotionStage;
    astPositionState: ARRAY[1..MotionConstants.MAX_STATE_MOTORS] OF ARRAY[1..GeneralConstants.MAX_STATES] OF ST_PositionState;
    afbInternal: ARRAY[1..2] OF FB_PositionStateInternal;
    nIter: UINT;
END_VAR


// Spoof motor enables
FOR nIter := 1 TO 3 DO
    astMotionStage[nIter].bAllEnable := TRUE;
    astMotionStage[nIter].bAllForwardEnable := TRUE;
    astMotionStage[nIter].bAllBackwardEnable := TRUE;
END_FOR
// Note: the fake motors show as position = 0, so they will be over/under the goals here
astPositionState[1][1].fPosition := 10;
astPositionState[1][1].fDelta := 1;
afbInternal[1](
    stMotionStage:=astMotionStage[1],
    stPositionState:=astPositionState[1][1],
);
SetGoodState(astPositionState[1][1]);

astPositionState[2][1].fPosition := -10;
astPositionState[2][1].fDelta := 1;
afbInternal[2](
    stMotionStage:=astMotionStage[2],
    stPositionState:=astPositionState[2][1],
);
SetGoodState(astPositionState[2][1]);

TestUnderOverGoals();
TestMaint();
TestCount();

METHOD TestCount
VAR_INST
    fbEnables: FB_StatePMPSEnablesND;
    fbFFHWO: FB_HardwareFFOutput := (bAutoReset := TRUE);
END_VAR

TEST('TestCount');

fbFFHWO.EvaluateOutput();
// No faults please
AssertTrue(
    fbFFHWO.q_xFastFaultOut,
    'Had faults prior to test',
);
fbEnables(
    astMotionStage:=astMotionStage,
    astPositionState:=astPositionState,
    fbFFHWO:=fbFFHWO,
    nGoalStateIndex:=1,
    sDeviceName:='TestUnderOverGoals',
    bMaintMode:=FALSE,
);
fbFFHWO.EvaluateOutput();
// Must fault with bad count
AssertFalse(
    fbFFHWO.q_xFastFaultOut,
    'Had no fault with bad count',
);

TEST_FINISHED();
END_METHOD

METHOD TestMaint
VAR_INST
    fbEnables: FB_StatePMPSEnablesND;
    fbFFHWO: FB_HardwareFFOutput := (bAutoReset := TRUE);
END_VAR

TEST('TestMaint');

fbFFHWO.EvaluateOutput();
// No faults please
AssertTrue(
    fbFFHWO.q_xFastFaultOut,
    'Had faults prior to test',
);
fbEnables(
    astMotionStage:=astMotionStage,
    astPositionState:=astPositionState,
    fbFFHWO:=fbFFHWO,
    nActiveMotorCount:=2,
    nGoalStateIndex:=1,
    sDeviceName:='TestUnderOverGoals',
    bMaintMode:=TRUE,
);
fbFFHWO.EvaluateOutput();
// Must fault in maint mode
AssertFalse(
    fbFFHWO.q_xFastFaultOut,
    'Had no fault in maintenance mode',
);
// All overrides should be relaxed
AssertTrue(
    fbEnables.abForwardEnabled[1],
    'In maintenance mode, we should be able to move anywhere',
);
AssertTrue(
    fbEnables.abBackwardEnabled[1],
    'In maintenance mode, we should be able to move anywhere',
);
AssertTrue(
    fbEnables.abForwardEnabled[1],
    'In maintenance mode, we should be able to move anywhere',
);
AssertTrue(
    fbEnables.abBackwardEnabled[1],
    'In maintenance mode, we should be able to move anywhere',
);

TEST_FINISHED();
END_METHOD

METHOD TestUnderOverGoals
VAR_INST
    fbEnables: FB_StatePMPSEnablesND;
    fbFFHWO: FB_HardwareFFOutput := (bAutoReset := TRUE);
END_VAR

TEST('TestUnderOverGoals');

IF NOT astPositionState[1][1].bUpdated OR NOT astPositionState[2][1].bUpdated THEN
    // Cannot run this test until the one-time-setup runs
    RETURN;
END_IF

fbEnables(
    astMotionStage:=astMotionStage,
    astPositionState:=astPositionState,
    fbFFHWO:=fbFFHWO,
    bEnable:=TRUE,
    nActiveMotorCount:=2,
    nGoalStateIndex:=1,
    sDeviceName:='TestUnderOverGoals',
    bMaintMode:=FALSE,
);
fbFFHWO.EvaluateOutput();
// No faults please
AssertTrue(
    fbFFHWO.q_xFastFaultOut,
    'Had faults in normal situation',
);
// All core enables are true
AssertTrue(
    astMotionStage[1].bAllForwardEnable,
    'Core enables should be TRUE',
);
AssertTrue(
    astMotionStage[1].bAllBackwardEnable,
    'Core enables should be TRUE',
);
AssertTrue(
    astMotionStage[2].bAllForwardEnable,
    'Core enables should be TRUE',
);
AssertTrue(
    astMotionStage[2].bAllBackwardEnable,
    'Core enables should be TRUE',
);
// But the overrides force us to move toward the goal
// Motor 1 is below the goal, Motor 2 is above the goal
AssertTrue(
    fbEnables.abForwardEnabled[1],
    'Motor 1 should be able to move up to the goal',
);
AssertFalse(
    fbEnables.abBackwardEnabled[1],
    'Motor 1 should not be able to move down away from the goal',
);
AssertFalse(
    fbEnables.abForwardEnabled[2],
    'Motor 2 should not be able to move up away from the goal',
);
AssertTrue(
    fbEnables.abBackwardEnabled[2],
    'Motor 2 should be able to move down to the goal',
);

TEST_FINISHED();
END_METHOD

END_FUNCTION_BLOCK

// Tests/FB_StateSetupHelper_Test
FUNCTION_BLOCK FB_StateSetupHelper_Test EXTENDS FB_TestSuite
VAR
    astStates: ARRAY[1..10] OF ST_PositionState;
    stDefaultDefault: ST_PositionState;
END_VAR


TestNormalCase();
TestDefaultOnly();
TestManyOverrides();
TestNoDefault();
TestOnlyOnce();

METHOD TestDefaultOnly
VAR
    fbStateSetup: FB_StateSetupHelper;
    stDefault: ST_PositionState := (
        sName := 'DEFAULT',
        fPosition := 100,
        nEncoderCount := 200,
        fDelta := 0.5,
        fVelocity := 10,
        fAccel := 12,
        fDecel := 24,
        bMoveOk := TRUE,
        bLocked := TRUE,
        bValid := TRUE,
        bUseRawCounts := TRUE
    );
    stOriginal: ST_PositionState;
    stTarget: ST_PositionState;
END_VAR

TEST('TestDefaultOnly');

// Add a pmps key
stDefault.stPMPS.sPmpsState := 'KEY';
// Cache the defaults to use as the check in case stDefault gets mutated by a bug
stOriginal := stDefault;
// Apply only defaults
fbStateSetup(stPositionState:=stDefault, bSetDefault:=TRUE);
fbStateSetup(stPositionState:=stTarget);
// Check everything
AssertEquals_STRING(stOriginal.sName, stTarget.sName, 'Wrong sName');
AssertEquals_LREAL(stOriginal.fPosition, stTarget.fPosition, 0, 'Wrong fPosition');
AssertEquals_UDINT(stOriginal.nEncoderCount, stTarget.nEncoderCount, 'Wrong nEncoderCount');
AssertEquals_LREAL(stOriginal.fDelta, stTarget.fDelta, 0, 'Wrong fDelta');
AssertEquals_LREAL(stOriginal.fVelocity, stTarget.fVelocity, 0, 'Wrong fVelocity');
AssertEquals_LREAL(stOriginal.fAccel, stTarget.fAccel, 0, 'Wrong fAccel');
AssertEquals_LREAL(stOriginal.fDecel, stTarget.fDecel, 0, 'Wrong fDecel');
AssertEquals_BOOL(stOriginal.bMoveOk, stTarget.bMoveOk, 'Wrong bMoveOk');
AssertEquals_BOOL(stOriginal.bLocked, stTarget.bLocked, 'Wrong bLocked');
AssertEquals_BOOL(stOriginal.bValid, stTarget.bValid, 'Wrong bValid');
AssertEquals_BOOL(stOriginal.bUseRawCounts, stTarget.bUseRawCounts, 'Wrong bUseRawCounts');
AssertEquals_STRING(stOriginal.stPMPS.sPmpsState, stTarget.stPMPS.sPmpsState, 'Wrong sPmpsState');

TEST_FINISHED();
END_METHOD

METHOD TestManyOverrides
VAR
    fbStateSetup: FB_StateSetupHelper;
    stDefault: ST_PositionState := (
        sName := 'POTATO',
        fPosition := 23,
        fDelta := 0.5,
        fVelocity := 10
    );
    stOne: ST_PositionState;
    stTwo: ST_PositionState;
END_VAR

TEST('TestManyOverrides');
// This is the case where the defaults are always overriden

fbStateSetup(stPositionState:=stDefault, bSetDefault:=TRUE);
fbStateSetup(stPositionState:=stOne, sName:='ONE', fPosition:=10, fDelta:=0.1, fVelocity:=20);
fbStateSetup(stPositionState:=stTWO, sName:='TWO', fPosition:=30, fDelta:=0.23, fVelocity:=4);

// Check Everything
AssertEquals_STRING('ONE', stOne.sName, 'Wrong sName in state 1');
AssertEquals_LREAL(10, stOne.fPosition, 0, 'Wrong fPosition in state 1');
AssertEquals_UDINT(stDefaultDefault.nEncoderCount, stOne.nEncoderCount, 'Wrong nEncoderCount in state 1');
AssertEquals_LREAL(0.1, stOne.fDelta, 0, 'Wrong fDelta in state 1');
AssertEquals_LREAL(20, stOne.fVelocity, 0, 'Wrong fVelocity in state 1');
AssertEquals_LREAL(stDefaultDefault.fAccel, stOne.fAccel, 0, 'Wrong fAccel in state 1');
AssertEquals_LREAL(stDefaultDefault.fDecel, stOne.fDecel, 0, 'Wrong fDecel in state 1');
AssertEquals_BOOL(stDefaultDefault.bMoveOk, stOne.bMoveOk, 'Wrong bMoveOk in state 1');
AssertEquals_BOOL(stDefaultDefault.bLocked, stOne.bLocked, 'Wrong bLocked in state 1');
AssertEquals_BOOL(stDefaultDefault.bValid, stOne.bValid, 'Wrong bValid in state 1');
AssertEquals_BOOL(stDefaultDefault.bUseRawCounts, stOne.bUseRawCounts, 'Wrong bUseRawCounts in state 1');
AssertEquals_STRING(stDefaultDefault.stPMPS.sPmpsState, stOne.stPMPS.sPmpsState, 'Wrong sPmpsState in state 1');

AssertEquals_STRING('TWO', stTwo.sName, 'Wrong sName in state 2');
AssertEquals_LREAL(30, stTwo.fPosition, 0, 'Wrong fPosition in state 2');
AssertEquals_UDINT(stDefaultDefault.nEncoderCount, stTwo.nEncoderCount, 'Wrong nEncoderCount in state 2');
AssertEquals_LREAL(0.23, stTwo.fDelta, 0, 'Wrong fDelta in state 2');
AssertEquals_LREAL(4, stTwo.fVelocity, 0, 'Wrong fVelocity in state 2');
AssertEquals_LREAL(stDefaultDefault.fAccel, stTwo.fAccel, 0, 'Wrong fAccel in state 2');
AssertEquals_LREAL(stDefaultDefault.fDecel, stTwo.fDecel, 0, 'Wrong fDecel in state 2');
AssertEquals_BOOL(stDefaultDefault.bMoveOk, stTwo.bMoveOk, 'Wrong bMoveOk in state 2');
AssertEquals_BOOL(stDefaultDefault.bLocked, stTwo.bLocked, 'Wrong bLocked in state 2');
AssertEquals_BOOL(stDefaultDefault.bValid, stTwo.bValid, 'Wrong bValid in state 2');
AssertEquals_BOOL(stDefaultDefault.bUseRawCounts, stTwo.bUseRawCounts, 'Wrong bUseRawCounts in state 2');
AssertEquals_STRING(stDefaultDefault.stPMPS.sPmpsState, stTwo.stPMPS.sPmpsState, 'Wrong sPmpsState in state 2');

TEST_FINISHED();
END_METHOD

METHOD TestNoDefault
VAR
    fbStateSetup: FB_StateSetupHelper;
    stTarget: ST_PositionState;
END_VAR

TEST('TestNoDefault');
// No default = invalid state + warning log message

fbStateSetup(stPositionState:=stTarget, sName:='TestNoDefault', sPmpsState:='TestPMPS', bValid:=TRUE);
// Only bValid matters, it must not be valid!
AssertFalse(stTarget.bValid, 'bValid should be FALSE with no default set.');

TEST_FINISHED();
END_METHOD

METHOD TestNormalCase
VAR
    fbStateSetup: FB_StateSetupHelper;
    stDefault: ST_PositionState;
END_VAR
VAR CONSTANT
    cDelta: LREAL := 0.5;
    cVelocity: LREAL := 10;
    cMoveOk: BOOL := TRUE;
    cValid: BOOL := TRUE;
END_VAR

TEST('TestNormalCase');
// Mimic what I might do in a real project

stDefault.fDelta := cDelta;
stDefault.fVelocity := cVelocity;
stDefault.bMoveOk := cMoveOk;
stDefault.bValid := cValid;

fbStateSetup(stPositionState:=stDefault, bSetDefault:=TRUE);
fbStateSetup(stPositionState:=astStates[1], sName:='OUT', fPosition:=10, sPmpsState:='FAKE_OUT');
fbStateSetup(stPositionState:=astStates[2], sName:='YAG', fPosition:=20, sPmpsState:='FAKE_YAG');
fbStateSetup(stPositionState:=astStates[3], sName:='TT', fPosition:=30, sPmpsState:='FAKE_TT');

// Check everything
AssertEquals_STRING('OUT', astStates[1].sName, 'Wrong sName in state 1');
AssertEquals_LREAL(10, astStates[1].fPosition, 0, 'Wrong fPosition in state 1');
AssertEquals_UDINT(stDefaultDefault.nEncoderCount, astStates[1].nEncoderCount, 'Wrong nEncoderCount in state 1');
AssertEquals_LREAL(cDelta, astStates[1].fDelta, 0, 'Wrong fDelta in state 1');
AssertEquals_LREAL(cVelocity, astStates[1].fVelocity, 0, 'Wrong fVelocity in state 1');
AssertEquals_LREAL(stDefaultDefault.fAccel, astStates[1].fAccel, 0, 'Wrong fAccel in state 1');
AssertEquals_LREAL(stDefaultDefault.fDecel, astStates[1].fDecel, 0, 'Wrong fDecel in state 1');
AssertEquals_BOOL(cMoveOk, astStates[1].bMoveOk, 'Wrong bMoveOk in state 1');
AssertEquals_BOOL(stDefaultDefault.bLocked, astStates[1].bLocked, 'Wrong bLocked in state 1');
AssertEquals_BOOL(cValid, astStates[1].bValid, 'Wrong bValid in state 1');
AssertEquals_BOOL(stDefaultDefault.bUseRawCounts, astStates[1].bUseRawCounts, 'Wrong bUseRawCounts in state 1');
AssertEquals_STRING('FAKE_OUT', astStates[1].stPMPS.sPmpsState, 'Wrong sPmpsState in state 1');

AssertEquals_STRING('YAG', astStates[2].sName, 'Wrong sName in state 2');
AssertEquals_LREAL(20, astStates[2].fPosition, 0, 'Wrong fPosition in state 2');
AssertEquals_UDINT(stDefaultDefault.nEncoderCount, astStates[2].nEncoderCount, 'Wrong nEncoderCount in state 2');
AssertEquals_LREAL(cDelta, astStates[2].fDelta, 0, 'Wrong fDelta in state 2');
AssertEquals_LREAL(cVelocity, astStates[2].fVelocity, 0, 'Wrong fVelocity in state 2');
AssertEquals_LREAL(stDefaultDefault.fAccel, astStates[2].fAccel, 0, 'Wrong fAccel in state 2');
AssertEquals_LREAL(stDefaultDefault.fDecel, astStates[2].fDecel, 0, 'Wrong fDecel in state 2');
AssertEquals_BOOL(cMoveOk, astStates[2].bMoveOk, 'Wrong bMoveOk in state 2');
AssertEquals_BOOL(stDefaultDefault.bLocked, astStates[2].bLocked, 'Wrong bLocked in state 2');
AssertEquals_BOOL(cValid, astStates[2].bValid, 'Wrong bValid in state 2');
AssertEquals_BOOL(stDefaultDefault.bUseRawCounts, astStates[2].bUseRawCounts, 'Wrong bUseRawCounts in state 2');
AssertEquals_STRING('FAKE_YAG', astStates[2].stPMPS.sPmpsState, 'Wrong sPmpsState in state 2');

AssertEquals_STRING('TT', astStates[3].sName, 'Wrong sName in state 3');
AssertEquals_LREAL(30, astStates[3].fPosition, 0, 'Wrong fPosition in state 3');
AssertEquals_UDINT(stDefaultDefault.nEncoderCount, astStates[3].nEncoderCount, 'Wrong nEncoderCount in state 3');
AssertEquals_LREAL(cDelta, astStates[3].fDelta, 0, 'Wrong fDelta in state 3');
AssertEquals_LREAL(cVelocity, astStates[3].fVelocity, 0, 'Wrong fVelocity in state 3');
AssertEquals_LREAL(stDefaultDefault.fAccel, astStates[3].fAccel, 0, 'Wrong fAccel in state 3');
AssertEquals_LREAL(stDefaultDefault.fDecel, astStates[3].fDecel, 0, 'Wrong fDecel in state 3');
AssertEquals_BOOL(cMoveOk, astStates[3].bMoveOk, 'Wrong bMoveOk in state 3');
AssertEquals_BOOL(stDefaultDefault.bLocked, astStates[3].bLocked, 'Wrong bLocked in state 3');
AssertEquals_BOOL(cValid, astStates[3].bValid, 'Wrong bValid in state 3');
AssertEquals_BOOL(stDefaultDefault.bUseRawCounts, astStates[3].bUseRawCounts, 'Wrong bUseRawCounts in state 3');
AssertEquals_STRING('FAKE_TT', astStates[3].stPMPS.sPmpsState, 'Wrong sPmpsState in state 3');

TEST_FINISHED();
END_METHOD

METHOD TestOnlyOnce
VAR
    fbStateSetup: FB_StateSetupHelper;
    stDefault: ST_PositionState;
    stTarget: ST_PositionState;
END_VAR

TEST('TestOnlyOnce');

// Required call, even though we don't need anything here
fbStateSetup(stPositionState:=stDefault, bSetDefault:=TRUE);
// Start with no position
AssertEquals_LREAL(stTarget.fPosition, 0, 0, 'Start position sanity check failed');
// Apply a new position
fbStateSetup(stPositionState:=stTarget, fPosition:=10);
AssertEquals_LREAL(stTarget.fPosition, 10, 0, 'Basic set position failed');
// Simulate the position state being used and updated via EPICS or otherwise
stTarget.bUpdated := TRUE; // Set by FB_PositionStateInternal
stTarget.fPosition := 12; // Someone tweaked the value in EPICS
// Run through the state setup again
fbStateSetup(stPositionState:=stTarget, fPosition:=10);
// But we should still be at position 12
AssertEquals_LREAL(stTarget.fPosition, 12, 0, 'FB_StateSetupHelper ran twice!');
// Unless we override the behavior
fbStateSetup(stPositionState:=stTarget, bForceUpdate:=TRUE, fPosition:=10);
AssertEquals_LREAL(stTarget.fPosition, 10, 0, 'bForceUpdate failed');

TEST_FINISHED();
END_METHOD

END_FUNCTION_BLOCK

// Tests/FB_TestStateInitTiming
FUNCTION_BLOCK FB_TestStateInitTiming EXTENDS TcUnit.FB_TestSuite
VAR
    stMotionStage: ST_MotionStage;
    fbMotionStageSim: FB_MotionStageSim;
END_VAR

fbMotionStageSim(
    stMotionStage:=stMotionStage,
    nEnableMode:=E_StageEnableMode.DURING_MOTION,
);

PassiveReinit();

METHOD PassiveReinit : BOOL
VAR_INPUT
END_VAR
VAR_INST
    fbStateSetup: FB_StateSetupHelper;
    stDefault: ST_PositionState := (
        fDelta := 0.5,
        fVelocity := 3,
        bMoveOk := TRUE,
        bValid := TRUE
    );
    eEnumSet: UINT;
    eEnumGet: UINT;
    stEpicsToPlc: ST_StateEpicsToPlc;
    stPlcToEpics: ST_StatePlcToEpics;
    fbCore: FB_PositionStateND_Core;
    astMotionStageMax: ARRAY[1..MotionConstants.MAX_STATE_MOTORS] OF ST_MotionStage;
    astPositionStateMax: ARRAY[1..MotionConstants.MAX_STATE_MOTORS] OF ARRAY[1..GeneralConstants.MAX_STATES] OF ST_PositionState;

    mcSetPos: MC_SetPosition;
    nCheckStep: UINT := 0;
    nFurthestStep: UINT;

    nLastState: UINT;
    nTransitionState: UINT := 99;
    nDoneState: UINT := 99;
    timer: TON;

    nSetPosErrCount: UINT := 0;
    nSetPosErrorID: UDINT;
END_VAR
TEST('PassiveReinit');

// State setup
fbStateSetup(stPositionState:=stDefault, bSetDefault:=TRUE);
fbStateSetup(stPositionState:=astPositionStateMax[1][1], sName:='ONE', fPosition:=10);
fbStateSetup(stPositionState:=astPositionStateMax[1][2], sName:='TWO', fPosition:=20);

// Run the state FB every cycle
astMotionStageMax[1] := stMotionStage;
fbCore(
    astMotionStageMax:=astMotionStageMax,
    astPositionStateMax:=astPositionStateMax,
    stEpicsToPlc:=stEpicsToPlc,
    stPlcToEpics:=stPlcToEpics,
    eEnumSet:=eEnumSet,
    eEnumGet:=eEnumGet,
    bEnable:=TRUE,
    nActiveMotorCount:=1,
);
stMotionStage := astMotionStageMax[1];

// Check and adjust different things as we go
CASE nCheckStep OF
    0:  // State begins at "Unknown", nCurrGoal begins at "Unknown"
        AssertEquals_UINT(
            Expected:=0,
            Actual:=eEnumGet,
            Message:='Did not start in unknown state',
        );
        AssertEquals_UINT(
            Expected:=0,
            Actual:=fbCore.nCurrGoal,
            Message:='Did not start with nCurrGoal unknown',
        );
        mcSetPos(
            Axis:=stMotionStage.Axis,
            Execute:=FALSE,
        );
        nCheckStep := 1;
    1:  // Set the current position to ONE/10
        mcSetPos(
            Axis:=stMotionStage.Axis,
            Execute:=TRUE,
            Position:=10,
        );
        IF mcSetPos.Done THEN
            mcSetPos(
                Axis:=stMotionStage.Axis,
                Execute:=FALSE,
            );
            nCheckStep := 2;
        ELSIF mcSetPos.Error THEN
            nSetPosErrCount := nSetPosErrCount + 1;
            nSetPosErrorID := mcSetPos.ErrorID;
            nCheckStep := 0;
        END_IF
    2:  // Without a move, the state and goal should both change to "ONE" if the position updates
        AssertEquals_UINT(
            Expected:=1,
            Actual:=eEnumGet,
            Message:='Read state did not change to ONE after setpos',
        );
        AssertEquals_UINT(
            Expected:=1,
            Actual:=fbCore.nCurrGoal,
            Message:='nCurrGoal did not change to ONE after setpos',
        );
        // Verify: no move requested
        AssertEquals_LREAL(
            Expected:=0,
            Actual:=stMotionStage.fPosition,
            Delta:=0.001,
            Message:='Set pos routine 1 actually gave us a move!',
        );
        nCheckStep := 3;
    3:  // Same as before, but to 20/TWO
        mcSetPos(
            Axis:=stMotionStage.Axis,
            Execute:=TRUE,
            Position:=20,
        );
        IF mcSetPos.Done THEN
            mcSetPos(
                Axis:=stMotionStage.Axis,
                Execute:=FALSE,
            );
            nCheckStep := 4;
        END_IF
    4:
        AssertEquals_UINT(
            Expected:=2,
            Actual:=eEnumGet,
            Message:='Read state did not change to TWO after setpos',
        );
        AssertEquals_UINT(
            Expected:=2,
            Actual:=fbCore.nCurrGoal,
            Message:='nCurrGoal did not change to TWO after setpos',
        );
        // Verify: no move requested
        AssertEquals_LREAL(
            Expected:=0,
            Actual:=stMotionStage.fPosition,
            Delta:=0.001,
            Message:='Set pos routine 2 actually gave us a move!',
        );
        nCheckStep := 5;
    5:  // Triggering a move should change the goal to the new state, without updating the readback
        eEnumSet := 1;
        nLastState := 2;
        nCheckStep := 6;
    6:
        AssertEquals_UINT(
            Expected:=1,
            Actual:=fbCore.nCurrGoal,
            Message:='nCurrGoal did not change to ONE in move',
        );
        // Looking for a readback transition 2 -> 0 -> 1
        // Record the next two transitions
        IF eEnumGet <> nLastState and nTransitionState = 99 THEN
            nTransitionState := eEnumGet;
        ELSIF eEnumGet <> nLastState and nDoneState = 99 THEN
            nDoneState := eEnumGet;
        END_IF
        nLastState := eEnumGet;
        IF stPlcToEpics.bDone THEN
            AssertEquals_UINT(
                Expected:=0,
                Actual:=nTransitionState,
                Message:='State did not transition 2 -> 0 in move',
            );
            AssertEquals_UINT(
                Expected:=1,
                Actual:=nDoneState,
                Message:='State did not transition 2 -> 0 -> 1 in move',
            );
            nCheckStep := 7;
        END_IF
    7: // The readback and curr goal should match after the move, then end test suite
        AssertEquals_UINT(
            Expected:=1,
            Actual:=eEnumGet,
            Message:='Read state did not change to ONE after move',
        );
        AssertEquals_UINT(
            Expected:=1,
            Actual:=fbCore.nCurrGoal,
            Message:='nCurrGoal did not stay at ONE after move',
        );
        AssertFalse(
            Condition:=timer.Q,
            Message:='Timeout in test',
        );
        TEST_FINISHED();
END_CASE

timer(IN:=TRUE, PT:=T#5s);
IF timer.Q THEN
    nCheckStep := 7;
END_IF
IF nCheckStep < 7 AND nFurthestStep < nCheckStep THEN
    nFurthestStep := nCheckStep;
END_IF
END_METHOD

END_FUNCTION_BLOCK

// Tests/PRG_TEST
PROGRAM PRG_TEST
VAR
    fb_TestHelperSetAndMove_Test: FB_TestHelperSetAndMove_Test;
    fb_AtPositionState_Test: FB_AtPositionState_Test;
    fb_PositionStateRead_Test: FB_PositionStateRead_Test;
    fb_PositionStateReadND_Test: FB_PositionStateReadND_Test;
    fb_PositionStateMove_Test: FB_PositionStateMove_Test;
    fb_PositionStateMoveND_Test: FB_PositionStateMoveND_Test;
    fb_PositionStateND_Test: FB_PositionStateND_Test;
    fb_NCErrorFFO_Test: FB_NCErrorFFO_Test;
    fb_MiscStatesErrorFFO_Test: FB_MiscStatesErrorFFO_Test;
    fb_MotionBPTM_Test: FB_MotionBPTM_Test;
    fb_MotionClearAsserts_Test: FB_MotionClearAsserts_Test;
    fb_StatePMPSEnables_Test: FB_StatePMPSEnables_Test;
    fb_MotionReadPMPSDBND_Test: FB_MotionReadPMPSDBND_Test;
    fb_PerMotorFFOND_Test: FB_PerMotorFFOND_Test;
    fb_StatePMPSEnablesND_Test: FB_StatePMPSEnablesND_Test;
    fb_PositionStatePMPSND_Test: FB_PositionStatePMPSND_Test;
    fb_StateSetupHelper_Test: FB_StateSetupHelper_Test;
    fb_TestStateInitTiming: FB_TestStateInitTiming;
    fb_AxisParameterSetExposed_Test: FB_AxisParameterSetExposed_Test;
END_VAR


TcUnit.RUN();

END_PROGRAM
